    16: (* Transition Delay After Last Bin (Bin 6) Closes *)
        Transition_Timer(IN := TRUE, PT := Step_Delay_Time);
        IF Transition_Timer.Q AND (NOT Discharge_Bin_Coarse[6] AND NOT Discharge_Bin_Fine[6]) THEN
            Transition_Timer(IN := FALSE);
            Step := 7; // Go to post-discharge wait step
        END_IF;

    7: (* Wait 2 Seconds After Closing the Last Bin *)
        Status_Message := 'Settling delay active';
        Completion_Timer(IN := TRUE, PT := Post_Complete_Delay);
        IF Completion_Timer.Q THEN
            Completion_Timer(IN := FALSE);
            Step := 8; // Proceed to reset last weight
        END_IF;
        
    8: (* Reset bin_last_weight to 0 & Complete *)
        bin_last_weight := 0.0;
        Sequence_Complete := TRUE;
        Status_Message := 'Sequence Completed';
        
        IF NOT Start_Button THEN
            Step := 0;
            Sequence_Complete := FALSE;
            Status_Message := 'System Idle';
            (* Reset all actual weights at completion once start is released *)
            FOR i := 1 TO 6 DO
                Actual_Weights[i] := 0.0;
            END_FOR;
        END_IF;
END_CASE;

END_PROGRAM

// PLC_AC500_V3/Application/old_version/Auto_Batching
FUNCTION_BLOCK Auto_Batching
VAR_INPUT
    Start_Button : BOOL;      // Signal to start the batching sequence
    E_Stop_Active : BOOL;     // Emergency Stop active signal
    load_cell_value : REAL;   // Weight value read from load cell
    Discharge_Bin_Feedback : ARRAY[1..6] OF BOOL; // Physical valve feedbacks
END_VAR
VAR_OUTPUT
    Auto_Bin : ARRAY[1..6] OF BOOL; // Motor/valve control outputs
    Actual_Weights : ARRAY[1..6] OF REAL; // Actual weight poured per silo
    Sequence_Complete : BOOL;  // Batch complete flag
END_VAR
VAR
    Step : INT := 0;          // State machine index (0: Idle, 1..6: Bins, 7: Delay, 8: Reset)
    bin_last_weight : REAL;   // Baseline weight on the load cell before starting current bin
    actual_bin : REAL;        // Current weight added from active bin
    target_act_bin : REAL;    // Target weight to add from the active bin
    bin_set_value : REAL;     // Setpoint weight for current active step
    
    (* Bin Mapping for 6 Auto Bins *)
    (* Maps physical Silo 1..6 to Material Index 1..20 *)
    Bin_Material_Index : ARRAY[1..6] OF INT := [
        1,   // Bin 1 maps to Material 1 (50.0 kg)
        2,   // Bin 2 maps to Material 2 (15.0 kg)
        0,   // Bin 3 is 0 (SKIPPED)
        4,   // Bin 4 maps to Material 4 (31.0 kg)
        5,   // Bin 5 maps to Material 5 (150.0 kg)
        6    // Bin 6 maps to Material 6 (10.0 kg)
    ];
    
    Mat_Idx : INT;
    i : INT;                  // General loop index
    
    (* TIMERS FOR TRANSITIONS & DELAYS *)
    Transition_Timer : TON;
    Completion_Timer : TON;
    Step_Delay_Time : TIME := T#2S;
    Post_Complete_Delay : TIME := T#2S;
    
    (* SELF-CONTAINED SIMULATION VARIABLES *)
    Simulation_Mode : BOOL := TRUE;
    Sim_Rate : REAL := 10.0;            // Simulated pouring speed (10.0 kg/s)
    Sim_Timer : TON;
    Start_Sim_Weight : REAL;
    Discharge_Active : BOOL;
END_VAR

(* Cumulative Gain-in-Weight Auto Batching FB *)

(* 1. SELF-CONTAINED SIMULATION WEIGHT MANAGEMENT *)
IF Simulation_Mode THEN
    (* Reset simulation to baseline (e.g. 2.0 kg) *)
    IF Step = 0 AND NOT Start_Button AND NOT Sequence_Complete THEN
        load_cell_value := 2.0;
        bin_last_weight := 2.0;
        Start_Sim_Weight := 2.0;
        Sim_Timer(IN := FALSE);
    END_IF;
    
    (* Check if any valve is actively discharging *)
    Discharge_Active := FALSE;
    IF Step >= 1 AND Step <= 6 THEN
        Discharge_Active := Auto_Bin[Step];
    END_IF;
    
    (* Simulate weight gain on the load cell *)
    IF Discharge_Active THEN
        Sim_Timer(IN := TRUE, PT := T#1000S);
        load_cell_value := Start_Sim_Weight + (TIME_TO_REAL(Sim_Timer.ET) / 1000.0) * Sim_Rate;
    ELSE
        Sim_Timer(IN := FALSE);
        Start_Sim_Weight := load_cell_value;
    END_IF;
END_IF;


(* 2. EMERGENCY STOP LOGIC *)
IF E_Stop_Active THEN
    FOR i := 1 TO 6 DO
        Auto_Bin[i] := FALSE;
        Actual_Weights[i] := 0.0;
    END_FOR;
    Sequence_Complete := FALSE;
    Step := 0;
    Transition_Timer(IN := FALSE);
    Completion_Timer(IN := FALSE);
    RETURN;
END_IF;


(* 3. RECIPE SEQUENCE START *)
IF Step = 0 AND Start_Button THEN
    Step := 1;
    bin_last_weight := load_cell_value;
    Sequence_Complete := FALSE;
    (* Clear actual weights on start *)
    FOR i := 1 TO 6 DO
        Actual_Weights[i] := 0.0;
    END_FOR;
END_IF;


(* 4. SEQUENCE CONTROL STATE MACHINE *)
CASE Step OF
    1..6: (* Discharging Silos 1 to 6 *)
        Mat_Idx := Bin_Material_Index[Step];
        
        IF Mat_Idx = 0 THEN
            (* Skip this bin instantly *)
            Step := Step + 1;
        ELSE
            (* Fetch target weight from global Recipe_Weights array *)
            bin_set_value := GVL.Recipe_Weights[Mat_Idx];
            target_act_bin := bin_set_value;
            
            (* Calculate weight added by current active bin *)
            actual_bin := load_cell_value - bin_last_weight;
            
            (* Update the actual weight in the array for the active bin *)
            Actual_Weights[Step] := actual_bin;
            
            (* Open discharge output valve *)
            Auto_Bin[Step] := TRUE;
            
            (* Check if target weight has been achieved *)
            IF actual_bin >= target_act_bin THEN
                Auto_Bin[Step] := FALSE;
                
                (* Set new baseline for the next step *)
                bin_last_weight := load_cell_value;
                
                (* Go to transition delay *)
                Step := 10 + Step; // Offset to separate transition states
            END_IF;
        END_IF;

    11..15: (* Transition Delays (Between Bins) *)
        Transition_Timer(IN := TRUE, PT := Step_Delay_Time);
        IF Transition_Timer.Q AND (NOT Auto_Bin[Step - 10] OR NOT Discharge_Bin_Feedback[Step - 10]) THEN
            Transition_Timer(IN := FALSE);
            Step := (Step - 10) + 1; // Advance to next bin
        END_IF;
        
    16: (* Transition Delay After Last Bin (Bin 6) Closes *)
        Transition_Timer(IN := TRUE, PT := Step_Delay_Time);
        IF Transition_Timer.Q AND (NOT Auto_Bin[6] OR NOT Discharge_Bin_Feedback[6]) THEN
            Transition_Timer(IN := FALSE);
            Step := 7; // Go to post-discharge wait step
        END_IF;

    7: (* Wait 2 Seconds After Closing the Last Bin *)
        Completion_Timer(IN := TRUE, PT := Post_Complete_Delay);
        IF Completion_Timer.Q THEN
            Completion_Timer(IN := FALSE);
            Step := 8; // Proceed to reset last weight
        END_IF;
        
    8: (* Reset bin_last_weight to 0 & Complete *)
        bin_last_weight := 0.0;
        Sequence_Complete := TRUE;
        
        IF NOT Start_Button THEN
            Step := 0;
            Sequence_Complete := FALSE;
            (* Reset all actual weights at completion once start is released *)
            FOR i := 1 TO 6 DO
                Actual_Weights[i] := 0.0;
            END_FOR;
        END_IF;
END_CASE;

END_FUNCTION_BLOCK

// PLC_AC500_V3/Application/old_version/Manual_Batching
FUNCTION_BLOCK Manual_Batching
VAR_INPUT
    Start_Button : BOOL;      // Signal to start the batching sequence
    E_Stop_Active : BOOL;     // Emergency Stop active signal
    load_cell_value : REAL;   // Weight value read from load cell
END_VAR
VAR_OUTPUT
    Manual_Bin : ARRAY[1..10] OF BOOL; // Prompts/indicators for Bins 7..16
    Actual_Weights : ARRAY[1..10] OF REAL; // Actual weight poured per silo
    Sequence_Complete : BOOL;  // Batch complete flag
END_VAR
VAR
    Step : INT := 0;          // State machine index (0: Idle, 1..10: Bins, 11..20: Delays, 30: Settling, 40: Complete)
    bin_last_weight : REAL;   // Baseline weight on the load cell before starting current bin
    actual_bin : REAL;        // Current weight added from active bin
    target_act_bin : REAL;    // Target weight to add from the active bin
    bin_set_value : REAL;     // Setpoint weight for current active step
    
    (* Bin Mapping for 10 Manual Bins *)
    (* Maps physical manual Silo 7..16 to Material Index 1..20 *)
    Bin_Manual_Index : ARRAY[1..10] OF INT := [
        7,    // Silo 7 maps to Material 7 (12.0 kg)
        8,    // Silo 8 maps to Material 8 (8.0 kg)
        0,    // Silo 9 is 0 (SKIPPED)
        10,   // Silo 10 maps to Material 10 (5.0 kg)
        11,   // Silo 11 maps to Material 11 (18.0 kg)
        12,   // Silo 12 maps to Material 12 (22.0 kg)
        13,   // Silo 13 maps to Material 13 (30.0 kg)
        14,   // Silo 14 maps to Material 14 (14.0 kg)
        15,   // Silo 15 maps to Material 15 (9.0 kg)
        16    // Silo 16 maps to Material 16 (11.0 kg)
    ];
    
    Mat_Idx : INT;
    i : INT;                  // General loop index
    
    (* TIMERS FOR TRANSITIONS & DELAYS *)
    Transition_Timer : TON;
    Completion_Timer : TON;
    Step_Delay_Time : TIME := T#2S;
    Post_Complete_Delay : TIME := T#2S;
    
    (* SELF-CONTAINED SIMULATION VARIABLES *)
    Simulation_Mode : BOOL := TRUE;
    Sim_Rate : REAL := 10.0;            // Simulated pouring speed (10.0 kg/s)
    Sim_Timer : TON;
    Start_Sim_Weight : REAL;
    Discharge_Active : BOOL;
END_VAR

(* Cumulative Gain-in-Weight Manual Batching FB (Simulates Operator Pouring) *)

(* 1. SIMULATION WEIGHT MANAGEMENT *)
IF Simulation_Mode THEN
    (* Reset simulation to baseline (e.g. 2.0 kg) *)
    IF Step = 0 AND NOT Start_Button AND NOT Sequence_Complete THEN
        load_cell_value := 2.0;
        bin_last_weight := 2.0;
        Start_Sim_Weight := 2.0;
        Sim_Timer(IN := FALSE);
    END_IF;
    
    (* Check if operator is actively pouring *)
    Discharge_Active := FALSE;
    IF Step >= 1 AND Step <= 10 THEN
        Discharge_Active := Manual_Bin[Step];
    END_IF;
    
    (* Simulate weight gain on the load cell *)
    IF Discharge_Active THEN
        Sim_Timer(IN := TRUE, PT := T#1000S);
        load_cell_value := Start_Sim_Weight + (TIME_TO_REAL(Sim_Timer.ET) / 1000.0) * Sim_Rate;
    ELSE
        Sim_Timer(IN := FALSE);
        Start_Sim_Weight := load_cell_value;
    END_IF;
END_IF;


(* 2. EMERGENCY STOP LOGIC *)
IF E_Stop_Active THEN
    FOR i := 1 TO 10 DO
        Manual_Bin[i] := FALSE;
        Actual_Weights[i] := 0.0;
    END_FOR;
    Sequence_Complete := FALSE;
    Step := 0;
    Transition_Timer(IN := FALSE);
    Completion_Timer(IN := FALSE);
    RETURN;
END_IF;


(* 3. RECIPE SEQUENCE START *)
IF Step = 0 AND Start_Button THEN
    Step := 1;
    bin_last_weight := load_cell_value;
    Sequence_Complete := FALSE;
    (* Clear actual weights on start *)
    FOR i := 1 TO 10 DO
        Actual_Weights[i] := 0.0;
    END_FOR;
END_IF;


(* 4. SEQUENCE CONTROL STATE MACHINE *)
CASE Step OF
    1..10: (* Prompts Silos 7 to 16 *)
        Mat_Idx := Bin_Manual_Index[Step];
        
        IF Mat_Idx = 0 THEN
            (* Skip this bin instantly *)
            Step := Step + 1;
        ELSE
            (* Fetch target weight from global Recipe_Weights array *)
            bin_set_value := GVL.Recipe_Weights[Mat_Idx];
            target_act_bin := bin_set_value;
            
            (* Calculate weight added by current active bin *)
            actual_bin := load_cell_value - bin_last_weight;
            
            (* Update the actual weight in the array for the active bin *)
            Actual_Weights[Step] := actual_bin;
            
            (* Prompt operator indicator active *)
            Manual_Bin[Step] := TRUE;
            
            (* Check if target weight has been achieved *)
            IF actual_bin >= target_act_bin THEN
                Manual_Bin[Step] := FALSE;
                
                (* Set new baseline for the next step *)
                bin_last_weight := load_cell_value;
                
                (* Go to transition delay *)
                Step := 10 + Step; // Offset to separate transition states
            END_IF;
        END_IF;

    11..19: (* Transition Delays (Between Bins) *)
        Transition_Timer(IN := TRUE, PT := Step_Delay_Time);
        IF Transition_Timer.Q THEN
            Transition_Timer(IN := FALSE);
            Step := (Step - 10) + 1; // Advance to next bin
        END_IF;
        
    20: (* Transition Delay After Last Bin (Bin 10) Closes *)
        Transition_Timer(IN := TRUE, PT := Step_Delay_Time);
        IF Transition_Timer.Q THEN
            Transition_Timer(IN := FALSE);
            Step := 30; // Go to post-discharge wait step (State 30)
        END_IF;

    30: (* Wait 2 Seconds After Closing the Last Bin *)
        Completion_Timer(IN := TRUE, PT := Post_Complete_Delay);
        IF Completion_Timer.Q THEN
            Completion_Timer(IN := FALSE);
            Step := 40; // Proceed to reset last weight (State 40)
        END_IF;
        
    40: (* Reset bin_last_weight to 0 & Complete *)
        bin_last_weight := 0.0;
        Sequence_Complete := TRUE;
        
        IF NOT Start_Button THEN
            Step := 0;
            Sequence_Complete := FALSE;
            (* Reset all actual weights at completion once start is released *)
            FOR i := 1 TO 10 DO
                Actual_Weights[i] := 0.0;
            END_FOR;
        END_IF;
END_CASE;

END_FUNCTION_BLOCK

// PLC_AC500_V3/Application/old_version/batching6
PROGRAM batching6
VAR
    Auto_Ctrl : Auto_Batching;
    Manual_Ctrl : Manual_Batching;
    
    (* Global Inputs & Toggles *)
    Start_Button : BOOL;
    E_Stop_Active : BOOL;
    
    (* Parallel Weight Feedbacks *)
    load_cell_auto : REAL;
    load_cell_manual : REAL;
    
    (* Process Outputs *)
    Auto_Bin : ARRAY[1..6] OF BOOL;
    Manual_Bin : ARRAY[1..10] OF BOOL;
    
    Auto_Weights : ARRAY[1..6] OF REAL;
    Manual_Weights : ARRAY[1..10] OF REAL;
    
    Auto_Complete : BOOL;
    Manual_Complete : BOOL;
    Sequence_Complete : BOOL;
END_VAR

(* Run Auto & Manual Batching pipelines concurrently in parallel *)

Auto_Ctrl(
    Start_Button := Start_Button,
    E_Stop_Active := E_Stop_Active,
    load_cell_value := load_cell_auto,
    Discharge_Bin_Feedback := ,
    Auto_Bin => Auto_Bin,
    Actual_Weights => Auto_Weights,
    Sequence_Complete => Auto_Complete
);

Manual_Ctrl(
    Start_Button := Start_Button,
    E_Stop_Active := E_Stop_Active,
    load_cell_value := load_cell_manual,
    Manual_Bin => Manual_Bin,
    Actual_Weights => Manual_Weights,
    Sequence_Complete => Manual_Complete
);

(* Global complete once both streams conclude *)
Sequence_Complete := Auto_Complete AND Manual_Complete;

END_PROGRAM

// PLC_AC500_V3/Application/old_version/Auto_Batching_V7
FUNCTION_BLOCK Auto_Batching_V7
VAR_INPUT
    Start_Button : BOOL;      // Signal to start the batching sequence
    E_Stop_Active : BOOL;     // Emergency Stop active signal
    load_cell_value : REAL;   // Weight value read from load cell
    Discharge_Bin_Feedback : ARRAY[1..6] OF BOOL; // Physical valve feedbacks
    Bin_Material_Index : ARRAY[1..6] OF INT;      // Mapped material index inputs
END_VAR
VAR_OUTPUT
    Auto_Bin : ARRAY[1..6] OF BOOL; // Motor/valve control outputs
    Actual_Weights : ARRAY[1..6] OF REAL; // Actual weight poured per silo
    Sequence_Complete : BOOL;  // Batch complete flag
    Active_Material_ID : INT;  // Currently active ingredient ID
    Active_Bin_ID : INT;       // Currently active physical Bin ID (1..6)
END_VAR
VAR
    Step : INT := 0;          // State machine index (0: Idle, 1..6: Bins, 7: Delay, 8: Reset)
    bin_last_weight : REAL;   // Baseline weight on the load cell before starting current bin
    actual_bin : REAL;        // Current weight added from active bin
    target_act_bin : REAL;    // Target weight to add from the active bin
    bin_set_value : REAL;     // Setpoint weight for current active step
    
    Mat_Idx : INT;
    i : INT;                  // General loop index
    
    (* TIMERS FOR TRANSITIONS & DELAYS *)
    Transition_Timer : TON;
    Completion_Timer : TON;
    Step_Delay_Time : TIME := T#2S;
    Post_Complete_Delay : TIME := T#2S;
    
    (* SELF-CONTAINED SIMULATION VARIABLES *)
    Simulation_Mode : BOOL := TRUE;
    Sim_Rate : REAL := 10.0;            // Simulated pouring speed (10.0 kg/s)
    Sim_Timer : TON;
    Start_Sim_Weight : REAL;
    Discharge_Active : BOOL;
END_VAR

(* Cumulative Gain-in-Weight Auto Batching FB V7 *)

(* 1. SELF-CONTAINED SIMULATION WEIGHT MANAGEMENT *)
IF Simulation_Mode THEN
    (* Reset simulation to baseline (e.g. 2.0 kg) *)
    IF Step = 0 AND NOT Start_Button AND NOT Sequence_Complete THEN
        load_cell_value := 2.0;
        bin_last_weight := 2.0;
        Start_Sim_Weight := 2.0;
        Sim_Timer(IN := FALSE);
    END_IF;
    
    (* Check if any valve is actively discharging *)
    Discharge_Active := FALSE;
    IF Step >= 1 AND Step <= 6 THEN
        Discharge_Active := Auto_Bin[Step];
    END_IF;
    
    (* Simulate weight gain on the load cell *)
    IF Discharge_Active THEN
        Sim_Timer(IN := TRUE, PT := T#1000S);
        load_cell_value := Start_Sim_Weight + (TIME_TO_REAL(Sim_Timer.ET) / 1000.0) * Sim_Rate;
    ELSE
        Sim_Timer(IN := FALSE);
        Start_Sim_Weight := load_cell_value;
    END_IF;
END_IF;


(* 2. EMERGENCY STOP LOGIC *)
IF E_Stop_Active THEN
    FOR i := 1 TO 6 DO
        Auto_Bin[i] := FALSE;
        Actual_Weights[i] := 0.0;
    END_FOR;
    Sequence_Complete := FALSE;
    Step := 0;
    Active_Material_ID := 0;
    Active_Bin_ID := 0;
    Transition_Timer(IN := FALSE);
    Completion_Timer(IN := FALSE);
    RETURN;
END_IF;


(* 3. RECIPE SEQUENCE START *)
IF Step = 0 AND Start_Button THEN
    Step := 1;
    bin_last_weight := load_cell_value;
    Sequence_Complete := FALSE;
    (* Clear actual weights on start *)
    FOR i := 1 TO 6 DO
        Actual_Weights[i] := 0.0;
    END_FOR;
END_IF;


(* 4. SEQUENCE CONTROL STATE MACHINE *)
CASE Step OF
    0:
        Active_Material_ID := 0;
        Active_Bin_ID := 0;
        
    1..6: (* Discharging Silos 1 to 6 *)
        Mat_Idx := Bin_Material_Index[Step];
        
        IF Mat_Idx = 0 THEN
            (* Skip this bin instantly *)
            Step := Step + 1;
        ELSE
            (* Fetch target weight from global Recipe_Weights array *)
            bin_set_value := GVL.Recipe_Weights[Mat_Idx];
            target_act_bin := bin_set_value;
            
            (* Calculate weight added by current active bin *)
            actual_bin := load_cell_value - bin_last_weight;
            
            (* Update the actual weight in the array for the active bin *)
            Actual_Weights[Step] := actual_bin;
            
            (* Open discharge output valve *)
            Auto_Bin[Step] := TRUE;
            
            (* Output currently active IDs *)
            Active_Material_ID := Mat_Idx;
            Active_Bin_ID := Step;
            
            (* Check if target weight has been achieved *)
            IF actual_bin >= target_act_bin THEN
                Auto_Bin[Step] := FALSE;
                
                (* Set new baseline for the next step *)
                bin_last_weight := load_cell_value;
                
                (* Go to transition delay *)
                Step := 10 + Step; // Offset to separate transition states
            END_IF;
        END_IF;

    11..15: (* Transition Delays (Between Bins) *)
        Active_Material_ID := 0;
        Active_Bin_ID := 0;
        Transition_Timer(IN := TRUE, PT := Step_Delay_Time);
        IF Transition_Timer.Q AND (NOT Auto_Bin[Step - 10] OR NOT Discharge_Bin_Feedback[Step - 10]) THEN
            Transition_Timer(IN := FALSE);
            Step := (Step - 10) + 1; // Advance to next bin
        END_IF;
        
    16: (* Transition Delay After Last Bin (Bin 6) Closes *)
        Active_Material_ID := 0;
        Active_Bin_ID := 0;
        Transition_Timer(IN := TRUE, PT := Step_Delay_Time);
        IF Transition_Timer.Q AND (NOT Auto_Bin[6] OR NOT Discharge_Bin_Feedback[6]) THEN
            Transition_Timer(IN := FALSE);
            Step := 7; // Go to post-discharge wait step
        END_IF;

    7: (* Wait 2 Seconds After Closing the Last Bin *)
        Active_Material_ID := 0;
        Active_Bin_ID := 0;
        Completion_Timer(IN := TRUE, PT := Post_Complete_Delay);
        IF Completion_Timer.Q THEN
            Completion_Timer(IN := FALSE);
            Step := 8; // Proceed to reset last weight
        END_IF;
        
    8: (* Reset bin_last_weight to 0 & Complete *)
        Active_Material_ID := 0;
        Active_Bin_ID := 0;
        bin_last_weight := 0.0;
        Sequence_Complete := TRUE;
        
        IF NOT Start_Button THEN
            Step := 0;
            Sequence_Complete := FALSE;
            (* Reset all actual weights at completion once start is released *)
            FOR i := 1 TO 6 DO
                Actual_Weights[i] := 0.0;
            END_FOR;
        END_IF;
END_CASE;

END_FUNCTION_BLOCK

// PLC_AC500_V3/Application/old_version/Manual_Batching_V7
FUNCTION_BLOCK Manual_Batching_V7
VAR_INPUT
    Start_Button : BOOL;      // Signal to start the batching sequence
    E_Stop_Active : BOOL;     // Emergency Stop active signal
    load_cell_value : REAL;   // Weight value read from load cell
    Bin_Manual_Index : ARRAY[1..10] OF INT; // Mapped material index inputs
END_VAR
VAR_OUTPUT
    Manual_Bin : ARRAY[1..10] OF BOOL; // Prompts/indicators for Bins 7..16
    Actual_Weights : ARRAY[1..10] OF REAL; // Actual weight poured per silo
    Sequence_Complete : BOOL;  // Batch complete flag
    Active_Material_ID : INT;  // Currently active ingredient ID
    Active_Bin_ID : INT;       // Currently active physical Bin ID (7..16)
END_VAR
VAR
    Step : INT := 0;          // State machine index (0: Idle, 1..10: Bins, 11..20: Delays, 30: Settling, 40: Complete)
    bin_last_weight : REAL;   // Baseline weight on the load cell before starting current bin
    actual_bin : REAL;        // Current weight added from active bin
    target_act_bin : REAL;    // Target weight to add from the active bin
    bin_set_value : REAL;     // Setpoint weight for current active step
    
    Mat_Idx : INT;
    i : INT;                  // General loop index
    
    (* TIMERS FOR TRANSITIONS & DELAYS *)
    Transition_Timer : TON;
    Completion_Timer : TON;
    Step_Delay_Time : TIME := T#2S;
    Post_Complete_Delay : TIME := T#2S;
    
    (* SELF-CONTAINED SIMULATION VARIABLES *)
    Simulation_Mode : BOOL := TRUE;
    Sim_Rate : REAL := 10.0;            // Simulated pouring speed (10.0 kg/s)
    Sim_Timer : TON;
    Start_Sim_Weight : REAL;
    Discharge_Active : BOOL;
END_VAR

(* Cumulative Gain-in-Weight Manual Batching FB V7 *)

(* 1. SIMULATION WEIGHT MANAGEMENT *)
IF Simulation_Mode THEN
    (* Reset simulation to baseline (e.g. 2.0 kg) *)
    IF Step = 0 AND NOT Start_Button AND NOT Sequence_Complete THEN
        load_cell_value := 2.0;
        bin_last_weight := 2.0;
        Start_Sim_Weight := 2.0;
        Sim_Timer(IN := FALSE);
    END_IF;
    
    (* Check if operator is actively pouring *)
    Discharge_Active := FALSE;
    IF Step >= 1 AND Step <= 10 THEN
        Discharge_Active := Manual_Bin[Step];
    END_IF;
    
    (* Simulate weight gain on the load cell *)
    IF Discharge_Active THEN
        Sim_Timer(IN := TRUE, PT := T#1000S);
        load_cell_value := Start_Sim_Weight + (TIME_TO_REAL(Sim_Timer.ET) / 1000.0) * Sim_Rate;
    ELSE
        Sim_Timer(IN := FALSE);
        Start_Sim_Weight := load_cell_value;
    END_IF;
END_IF;


(* 2. EMERGENCY STOP LOGIC *)
IF E_Stop_Active THEN
    FOR i := 1 TO 10 DO
        Manual_Bin[i] := FALSE;
        Actual_Weights[i] := 0.0;
    END_FOR;
    Sequence_Complete := FALSE;
    Step := 0;
    Active_Material_ID := 0;
    Active_Bin_ID := 0;
    Transition_Timer(IN := FALSE);
    Completion_Timer(IN := FALSE);
    RETURN;
END_IF;


(* 3. RECIPE SEQUENCE START *)
IF Step = 0 AND Start_Button THEN
    Step := 1;
    bin_last_weight := load_cell_value;
    Sequence_Complete := FALSE;
    (* Clear actual weights on start *)
    FOR i := 1 TO 10 DO
        Actual_Weights[i] := 0.0;
    END_FOR;
END_IF;


(* 4. SEQUENCE CONTROL STATE MACHINE *)
CASE Step OF
    0:
        Active_Material_ID := 0;
        Active_Bin_ID := 0;
        
    1..10: (* Prompts Silos 7 to 16 *)
        Mat_Idx := Bin_Manual_Index[Step];
        
        IF Mat_Idx = 0 THEN
            (* Skip this bin instantly *)
            Step := Step + 1;
        ELSE
            (* Fetch target weight from global Recipe_Weights array *)
            bin_set_value := GVL.Recipe_Weights[Mat_Idx];
            target_act_bin := bin_set_value;
            
            (* Calculate weight added by current active bin *)
            actual_bin := load_cell_value - bin_last_weight;
            
            (* Update the actual weight in the array for the active bin *)
            Actual_Weights[Step] := actual_bin;
            
            (* Prompt operator indicator active *)
            Manual_Bin[Step] := TRUE;
            
            (* Output currently active IDs (Shift to physical Silo ID 7..16) *)
            Active_Material_ID := Mat_Idx;
            Active_Bin_ID := Step;
            
            (* Check if target weight has been achieved *)
            IF actual_bin >= target_act_bin THEN
                Manual_Bin[Step] := FALSE;
                
                (* Set new baseline for the next step *)
                bin_last_weight := load_cell_value;
                
                (* Go to transition delay *)
                Step := 10 + Step; // Offset to separate transition states
            END_IF;
        END_IF;

    11..19: (* Transition Delays (Between Bins) *)
        Active_Material_ID := 0;
        Active_Bin_ID := 0;
        Transition_Timer(IN := TRUE, PT := Step_Delay_Time);
        IF Transition_Timer.Q THEN
            Transition_Timer(IN := FALSE);
            Step := (Step - 10) + 1; // Advance to next bin
        END_IF;
        
    20: (* Transition Delay After Last Bin (Bin 10) Closes *)
        Active_Material_ID := 0;
        Active_Bin_ID := 0;
        Transition_Timer(IN := TRUE, PT := Step_Delay_Time);
        IF Transition_Timer.Q THEN
            Transition_Timer(IN := FALSE);
            Step := 30; // Go to post-discharge wait step (State 30)
        END_IF;

    30: (* Wait 2 Seconds After Closing the Last Bin *)
        Active_Material_ID := 0;
        Active_Bin_ID := 0;
        Completion_Timer(IN := TRUE, PT := Post_Complete_Delay);
        IF Completion_Timer.Q THEN
            Completion_Timer(IN := FALSE);
            Step := 40; // Proceed to reset last weight (State 40)
        END_IF;
        
    40: (* Reset bin_last_weight to 0 & Complete *)
        Active_Material_ID := 0;
        Active_Bin_ID := 0;
        bin_last_weight := 0.0;
        Sequence_Complete := TRUE;
        
        IF NOT Start_Button THEN
            Step := 0;
            Sequence_Complete := FALSE;
            (* Reset all actual weights at completion once start is released *)
            FOR i := 1 TO 10 DO
                Actual_Weights[i] := 0.0;
            END_FOR;
        END_IF;
END_CASE;

END_FUNCTION_BLOCK

// PLC_AC500_V3/Application/old_version/batching7
PROGRAM batching7
VAR
    Auto_Ctrl : Auto_Batching_V7;
    Manual_Ctrl : Manual_Batching_V7;
    
    (* Global Inputs & Toggles *)
    Start_Button : BOOL;
    E_Stop_Active : BOOL;
    
    (* Parallel Weight Feedbacks *)
    load_cell_auto : REAL;
    load_cell_manual : REAL;
    
    (* Process Outputs *)
    Auto_Bin : ARRAY[1..6] OF BOOL;
    Manual_Bin : ARRAY[1..10] OF BOOL;
    
    Auto_Weights : ARRAY[1..6] OF REAL;
    Manual_Weights : ARRAY[1..10] OF REAL;
    
    Auto_Complete : BOOL;
    Manual_Complete : BOOL;
    Sequence_Complete : BOOL;
    
    (* Cross-Validation *)
    Error_Code : INT := 0; // 0 = OK, 1 = Duplicate Material ID detected
    Status_Message : STRING := 'System Ready';
    
    (* Arrays defined here to allow check before FB execution *)
    Bin_Material_Index : ARRAY[1..6] OF INT := [1, 2, 0, 4, 5, 6];
    Bin_Manual_Index : ARRAY[1..10] OF INT := [7, 8, 0, 10, 11, 12, 13, 14, 15, 16];
    
    (* Active IDs as integer monitors *)
    Auto_Active_Mat : INT;
    Auto_Active_Bin : INT;
    Manual_Active_Mat : INT;
    Manual_Active_Bin : INT;
    
    i : INT;
    j : INT;
    Duplicate_Found : BOOL;
END_VAR

(* 1. CROSS-ARRAY DISTINCT MATERIAL VALIDATION *)
Duplicate_Found := FALSE;
FOR i := 1 TO 6 DO
    IF Bin_Material_Index[i] <> 0 THEN
        FOR j := 1 TO 10 DO
            IF Bin_Material_Index[i] = Bin_Manual_Index[j] THEN
                Duplicate_Found := TRUE;
            END_IF;
        END_FOR;
    END_IF;
END_FOR;

IF Duplicate_Found THEN
    Error_Code := 1;
    Status_Message := 'Error 1: Duplicate Material ID in Auto and Manual tables!';
    
    (* Shut off all outputs and abort execution *)
    FOR i := 1 TO 6 DO Auto_Bin[i] := FALSE; END_FOR;
    FOR i := 1 TO 10 DO Manual_Bin[i] := FALSE; END_FOR;
    
    (* Reset control blocks *)
    Auto_Ctrl(Start_Button := FALSE, E_Stop_Active := TRUE);
    Manual_Ctrl(Start_Button := FALSE, E_Stop_Active := TRUE);
    RETURN;
ELSE
    Error_Code := 0;
END_IF;

(* 2. EXECUTION OF BATCH CONTROLLERS *)
Auto_Ctrl(
    Start_Button := Start_Button,
    E_Stop_Active := E_Stop_Active,
    load_cell_value := load_cell_auto,
    Bin_Material_Index := Bin_Material_Index,
    Auto_Bin => Auto_Bin,
    Actual_Weights => Auto_Weights,
    Sequence_Complete => Auto_Complete,
    Active_Material_ID => Auto_Active_Mat,
    Active_Bin_ID => Auto_Active_Bin
);

Manual_Ctrl(
    Start_Button := Start_Button,
    E_Stop_Active := E_Stop_Active,
    load_cell_value := load_cell_manual,
    Bin_Manual_Index := Bin_Manual_Index,
    Manual_Bin => Manual_Bin,
    Actual_Weights => Manual_Weights,
    Sequence_Complete => Manual_Complete,
    Active_Material_ID => Manual_Active_Mat,
    Active_Bin_ID => Manual_Active_Bin
);

Sequence_Complete := Auto_Complete AND Manual_Complete;

IF Sequence_Complete THEN
    Status_Message := 'Batch Completed';
ELSIF Start_Button THEN
    Status_Message := 'Batch In Progress';
ELSE
    Status_Message := 'System Ready';
END_IF;

END_PROGRAM

// PLC_AC500_V3/Application/old_version/Auto_Batching_V8
FUNCTION_BLOCK Auto_Batching_V8
VAR_INPUT
    Start_Button : BOOL;      // Signal to start the batching sequence
    E_Stop_Active : BOOL;     // Emergency Stop active signal
    Discharge_Bin_Feedback : ARRAY[1..6] OF BOOL; // Physical valve feedbacks
    Auto_Bin_Material_Mapping : ARRAY[1..6] OF INT; // Material index mapping for 6 bins
    Auto_Coarse_To_Fine_speed : ARRAY[1..6] OF REAL; // Cutoff weight thresholds (kg)
END_VAR
VAR_IN_OUT
    load_cell_value : REAL;   // Weight value read/written from load cell
END_VAR
VAR_OUTPUT
    Auto_Bin : ARRAY[1..6] OF BOOL; // Coarse feed valve outputs
    auto_bin_cutoff : ARRAY[1..6] OF BOOL; // Fine feed cutoff trigger indicators
    auto_bin_motor : ARRAY[1..6] OF BOOL; // Main conveyor motor outputs
    Actual_Weights : ARRAY[1..6] OF REAL; // Actual weight poured per silo
    Sequence_Complete : BOOL;  // Batch complete flag
    Active_Material_ID : INT;  // Currently active ingredient ID
    Active_Bin_ID : INT;       // Currently active physical Bin ID (1..6)
    Active_Target_Weight : REAL; // Recipe target weight of active bin
    Error_Code : INT;          // Active error code
    Status_Message : STRING;   // Diagnostic text message
END_VAR
VAR
    Step : INT := 0;          // State machine index (0: Idle, 1..6: Bins, 11..16: Delays, 7: Settling, 8: Complete, 99: Error)
    bin_last_weight : REAL;   // Baseline weight on the load cell before starting current bin
    actual_bin : REAL;        // Current weight added from active bin
    target_act_bin : REAL;    // Target weight to add from the active bin
    bin_set_value : REAL;     // Setpoint weight for current active step
    cutoff_trigger_weight : REAL; // Calculated target threshold weight minus cutoff value
    
    Mat_Idx : INT;
    i : INT;                  // General loop index
    
    (* TIMERS FOR TRANSITIONS & DELAYS *)
    Transition_Timer : TON;
    Completion_Timer : TON;
    Step_Delay_Time : TIME := T#2S;
    Post_Complete_Delay : TIME := T#2S;
    
    (* SELF-CONTAINED SIMULATION VARIABLES *)
    Simulation_Mode : BOOL := TRUE;
    Sim_Rate : REAL := 10.0;            // Simulated pouring speed (10.0 kg/s)
    Sim_Timer : TON;
    Start_Sim_Weight : REAL;
    Discharge_Active : BOOL;
END_VAR

(* Auto Batching FB V8 matching batching7 sequence exactly *)

(* 1. SELF-CONTAINED SIMULATION WEIGHT MANAGEMENT *)
IF Simulation_Mode AND Step <> 99 THEN
    (* Reset simulation to baseline *)
    IF Step = 0 AND NOT Start_Button AND NOT Sequence_Complete THEN
        load_cell_value := 0.0;
        bin_last_weight := 0.0;
        Start_Sim_Weight := 0.0;
        Sim_Timer(IN := FALSE);
    END_IF;
    
    (* Check if any valve is actively discharging *)
    Discharge_Active := FALSE;
    IF Step >= 1 AND Step <= 6 THEN
        Discharge_Active := auto_bin_motor[Step];
    END_IF;
    
    (* Simulate weight gain on the load cell *)
    IF Discharge_Active THEN
        Sim_Timer(IN := TRUE, PT := T#1000S);
        load_cell_value := Start_Sim_Weight + (TIME_TO_REAL(Sim_Timer.ET) / 1000.0) * Sim_Rate;
    ELSE
        Sim_Timer(IN := FALSE);
        Start_Sim_Weight := load_cell_value;
    END_IF;
END_IF;


(* 2. EMERGENCY STOP LOGIC (Error 12) *)
IF E_Stop_Active THEN
    FOR i := 1 TO 6 DO
        Auto_Bin[i] := FALSE;
        auto_bin_cutoff[i] := FALSE;
        auto_bin_motor[i] := FALSE;
    END_FOR;
    Sequence_Complete := FALSE;
    Active_Material_ID := 0;
    Active_Bin_ID := 0;
    Active_Target_Weight := 0.0;
    Error_Code := 12;
    Status_Message := 'Error 12: Emergency Stop Active!';
    Step := 99;
    Transition_Timer(IN := FALSE);
    Completion_Timer(IN := FALSE);
    RETURN;
END_IF;


(* 3. RECIPE SEQUENCE START *)
IF Step = 0 AND Start_Button THEN
    Step := 1;
    bin_last_weight := load_cell_value;
    Sequence_Complete := FALSE;
    Error_Code := 0;
    Status_Message := 'Auto Batch Started';
    Active_Target_Weight := 0.0;
    (* Clear actual weights and outputs on start *)
    FOR i := 1 TO 6 DO
        Actual_Weights[i] := 0.0;
        Auto_Bin[i] := FALSE;
        auto_bin_cutoff[i] := FALSE;
        auto_bin_motor[i] := FALSE;
    END_FOR;
END_IF;


(* 4. SEQUENCE CONTROL STATE MACHINE *)
CASE Step OF
    0:
        Active_Material_ID := 0;
        Active_Bin_ID := 0;
        Active_Target_Weight := 0.0;
        IF Error_Code = 0 THEN Status_Message := 'Auto Idle'; END_IF;
        
    1..6: (* Discharging Silos 1 to 6 *)
        Mat_Idx := Auto_Bin_Material_Mapping[Step];
        
        IF Mat_Idx = 0 THEN
            (* Skip this bin instantly *)
            Step := Step + 1;
        ELSE
            (* Fetch target weight from global Recipe_Weights array *)
            bin_set_value := GVL.Recipe_Weights[Mat_Idx];
            target_act_bin := bin_set_value;
            Active_Target_Weight := target_act_bin;
            
            (* Calculate weight added by current active bin *)
            actual_bin := load_cell_value - bin_last_weight;
            Actual_Weights[Step] := actual_bin;
            
            (* Get cutoff threshold *)
            cutoff_trigger_weight := target_act_bin - Auto_Coarse_To_Fine_speed[Step];
            
            Active_Material_ID := Mat_Idx;
            Active_Bin_ID := Step;
            Status_Message := 'Auto Pouring';
            
            (* COARSE/FINE FEED TRANSITIONS *)
            IF actual_bin < cutoff_trigger_weight THEN
                (* Phase 1: Coarse Feed (Conveyor Motor ON, Main Valve ON, Fine Cutoff OFF) *)
                Auto_Bin[Step] := TRUE;
                auto_bin_cutoff[Step] := FALSE;
                auto_bin_motor[Step] := TRUE;
            ELSIF actual_bin < target_act_bin THEN
                (* Phase 2: Fine Feed (Conveyor Motor ON, Main Valve OFF, Fine Cutoff ON) *)
                Auto_Bin[Step] := FALSE;
                auto_bin_cutoff[Step] := TRUE;
                auto_bin_motor[Step] := TRUE;
            ELSE
                (* Phase 3: Completed (All OFF) *)
                Auto_Bin[Step] := FALSE;
                auto_bin_cutoff[Step] := FALSE;
                auto_bin_motor[Step] := FALSE;
                bin_last_weight := load_cell_value;
                Active_Target_Weight := 0.0;
                Step := 10 + Step; // Offset to separate transition states
            END_IF;
            
            (* RUNTIME CHECKS *)
            (* Check 21 & 22: Scale Limits *)
            IF load_cell_value > 500.0 THEN
                Error_Code := 21;
                Status_Message := 'Error 21: Scale Overloaded!';
                Step := 99;
                RETURN;
            ELSIF load_cell_value < 0.0 THEN
                Error_Code := 22;
                Status_Message := 'Error 22: Scale Underloaded/Fault!';
                Step := 99;
                RETURN;
            END_IF;
        END_IF;

    11..15: (* Transition Delays (Between Bins) *)
        Active_Material_ID := 0;
        Active_Bin_ID := 0;
        Active_Target_Weight := 0.0;
        Status_Message := 'Transition Delay';
        
        Transition_Timer(IN := TRUE, PT := Step_Delay_Time);
        IF Transition_Timer.Q THEN
            Transition_Timer(IN := FALSE);
            Step := (Step - 10) + 1; // Advance to next bin
        END_IF;
        
    16: (* Transition Delay After Last Bin (Bin 6) Closes *)
        Active_Material_ID := 0;
        Active_Bin_ID := 0;
        Active_Target_Weight := 0.0;
        Status_Message := 'Settling Last Bin';
        
        Transition_Timer(IN := TRUE, PT := Step_Delay_Time);
        IF Transition_Timer.Q THEN
            Transition_Timer(IN := FALSE);
            Step := 7; // Go to post-discharge wait step
        END_IF;

    7: (* Wait 2 Seconds After Closing the Last Bin *)
        Active_Material_ID := 0;
        Active_Bin_ID := 0;
        Active_Target_Weight := 0.0;
        Status_Message := 'Settling Delay';
        Completion_Timer(IN := TRUE, PT := Post_Complete_Delay);
        IF Completion_Timer.Q THEN
            Completion_Timer(IN := FALSE);
            Step := 8; // Proceed to reset last weight
        END_IF;
        
    8: (* Reset bin_last_weight to 0 & Complete *)
        Active_Material_ID := 0;
        Active_Bin_ID := 0;
        Active_Target_Weight := 0.0;
        Status_Message := 'Sequence Completed';
        bin_last_weight := 0.0;
        Sequence_Complete := TRUE;
        
        IF NOT Start_Button THEN
            Step := 0;
            Sequence_Complete := FALSE;
            (* Reset all actual weights at completion once start is released *)
            FOR i := 1 TO 6 DO
                Actual_Weights[i] := 0.0;
            END_FOR;
        END_IF;
        
    99: (* Error Abort state *)
        FOR i := 1 TO 6 DO 
            Auto_Bin[i] := FALSE; 
            auto_bin_cutoff[i] := FALSE;
            auto_bin_motor[i] := FALSE;
        END_FOR;
        Active_Material_ID := 0;
        Active_Bin_ID := 0;
        Active_Target_Weight := 0.0;
        IF NOT Start_Button THEN
            Step := 0;
            Error_Code := 0;
            Status_Message := 'Auto Idle';
        END_IF;
END_CASE;

END_FUNCTION_BLOCK

// PLC_AC500_V3/Application/old_version/Manual_Batching_V8
FUNCTION_BLOCK Manual_Batching_V8
VAR_INPUT
    Start_Button : BOOL;      // Signal to start the batching sequence
    E_Stop_Active : BOOL;     // Emergency Stop active signal
    Manual_Bin_Material_Mapping : ARRAY[1..10] OF INT; // Material index mapping for 10 manual silos
    Manual_Coarse_To_Fine_speed : ARRAY[1..10] OF REAL; // Cutoff weight thresholds (kg)
END_VAR
VAR_IN_OUT
    load_cell_value : REAL;   // Weight value read/written from load cell
END_VAR
VAR_OUTPUT
    Manual_Bin : ARRAY[1..10] OF BOOL; // Prompts/indicators for Bins 7..16
    manual_bin_cutoff : ARRAY[1..10] OF BOOL; // Manual pre-cutoff indicators
    manual_bin_motor : ARRAY[1..10] OF BOOL; // Main manual feeder motor outputs
    Actual_Weights : ARRAY[1..10] OF REAL; // Actual weight poured per silo
    Sequence_Complete : BOOL;  // Batch complete flag
    Active_Material_ID : INT;  // Currently active ingredient ID
    Active_Bin_ID : INT;       // Currently active physical Bin ID (7..16)
    Active_Target_Weight : REAL; // Recipe target weight of active bin
    Error_Code : INT;          // Active error code
    Status_Message : STRING;   // Diagnostic text message
END_VAR
VAR
    Step : INT := 0;          // State machine index (0: Idle, 1..10: Bins, 11..20: Delays, 30: Settling, 40: Complete, 99: Error)
    bin_last_weight : REAL;   // Baseline weight on the load cell before starting current bin
    actual_bin : REAL;        // Current weight added from active bin
    target_act_bin : REAL;    // Target weight to add from the active bin
    bin_set_value : REAL;     // Setpoint weight for current active step
    cutoff_trigger_weight : REAL; // Calculated target threshold weight minus cutoff value
    
    Mat_Idx : INT;
    i : INT;                  // General loop index
    
    (* TIMERS FOR TRANSITIONS & DELAYS *)
    Transition_Timer : TON;
    Completion_Timer : TON;
    Step_Delay_Time : TIME := T#2S;
    Post_Complete_Delay : TIME := T#2S;
    
    (* DIAGNOSTIC TIMERS *)
    Operator_Timer : TON;
    
    (* SELF-CONTAINED SIMULATION VARIABLES *)
    Simulation_Mode : BOOL := TRUE;
    Sim_Rate : REAL := 10.0;            // Simulated pouring speed (10.0 kg/s)
    Sim_Timer : TON;
    Start_Sim_Weight : REAL;
    Discharge_Active : BOOL;
END_VAR

(* Manual Batching FB V8 with Diagnostic Error Checks *)

(* 1. SIMULATION WEIGHT MANAGEMENT *)
IF Simulation_Mode AND Step <> 99 THEN
    (* Reset simulation to baseline *)
    IF Step = 0 AND NOT Start_Button AND NOT Sequence_Complete THEN
        load_cell_value := 0.0;
        bin_last_weight := 0.0;
        Start_Sim_Weight := 0.0;
        Sim_Timer(IN := FALSE);
    END_IF;
    
    (* Check if operator is actively pouring *)
    Discharge_Active := FALSE;
    IF Step >= 1 AND Step <= 10 THEN
        Discharge_Active := manual_bin_motor[Step];
    END_IF;
    
    (* Simulate weight gain on the load cell *)
    IF Discharge_Active THEN
        Sim_Timer(IN := TRUE, PT := T#1000S);
        load_cell_value := Start_Sim_Weight + (TIME_TO_REAL(Sim_Timer.ET) / 1000.0) * Sim_Rate;
    ELSE
        Sim_Timer(IN := FALSE);
        Start_Sim_Weight := load_cell_value;
    END_IF;
END_IF;


(* 2. EMERGENCY STOP LOGIC (Error 12) *)
IF E_Stop_Active THEN
    FOR i := 1 TO 10 DO
        Manual_Bin[i] := FALSE;
        manual_bin_cutoff[i] := FALSE;
        manual_bin_motor[i] := FALSE;
    END_FOR;
    Sequence_Complete := FALSE;
    Active_Material_ID := 0;
    Active_Bin_ID := 0;
    Active_Target_Weight := 0.0;
    Error_Code := 12;
    Status_Message := 'Error 12: Emergency Stop Active!';
    Step := 99;
    Transition_Timer(IN := FALSE);
    Completion_Timer(IN := FALSE);
    RETURN;
END_IF;


(* 3. RECIPE SEQUENCE START *)
IF Step = 0 AND Start_Button THEN
    Step := 1;
    bin_last_weight := load_cell_value;
    Sequence_Complete := FALSE;
    Error_Code := 0;
    Status_Message := 'Manual Batch Started';
    Active_Target_Weight := 0.0;
    (* Clear actual weights on start *)
    FOR i := 1 TO 10 DO
        Actual_Weights[i] := 0.0;
        Manual_Bin[i] := FALSE;
        manual_bin_cutoff[i] := FALSE;
        manual_bin_motor[i] := FALSE;
    END_FOR;
END_IF;


(* 4. SEQUENCE CONTROL STATE MACHINE *)
CASE Step OF
    0:
        Active_Material_ID := 0;
        Active_Bin_ID := 0;
        Active_Target_Weight := 0.0;
        IF Error_Code = 0 THEN Status_Message := 'Manual Idle'; END_IF;
        
    1..10: (* Prompts Silos 7 to 16 *)
        Mat_Idx := Manual_Bin_Material_Mapping[Step];
        
        IF Mat_Idx = 0 THEN
            (* Skip this bin instantly *)
            Step := Step + 1;
        ELSE
            (* Fetch target weight from global Recipe_Weights array *)
            bin_set_value := GVL.Recipe_Weights[Mat_Idx];
            target_act_bin := bin_set_value;
            Active_Target_Weight := target_act_bin;
            
            (* Calculate weight added by current active bin *)
            actual_bin := load_cell_value - bin_last_weight;
            Actual_Weights[Step] := actual_bin;
            
            (* Get cutoff threshold *)
            cutoff_trigger_weight := target_act_bin - Manual_Coarse_To_Fine_speed[Step];
            
            Active_Material_ID := Mat_Idx;
            Active_Bin_ID := Step;
            Status_Message := 'Manual Pouring Active';
            
            (* COARSE/FINE FEED TRANSITIONS *)
            IF actual_bin < cutoff_trigger_weight THEN
                (* Phase 1: Coarse Feed (Motor ON, Prompt ON, Cutoff OFF) *)
                Manual_Bin[Step] := TRUE;
                manual_bin_cutoff[Step] := FALSE;
                manual_bin_motor[Step] := TRUE;
            ELSIF actual_bin < target_act_bin THEN
                (* Phase 2: Fine Feed (Motor ON, Prompt OFF, Cutoff ON) *)
                Manual_Bin[Step] := FALSE;
                manual_bin_cutoff[Step] := TRUE;
                manual_bin_motor[Step] := TRUE;
            ELSE
                (* Phase 3: Completed (All OFF) *)
                Manual_Bin[Step] := FALSE;
                manual_bin_cutoff[Step] := FALSE;
                manual_bin_motor[Step] := FALSE;
                bin_last_weight := load_cell_value;
                Active_Target_Weight := 0.0;
                Step := 10 + Step; // Offset to separate transition states
            END_IF;
            
            (* RUNTIME CHECKS *)
            (* Check 21 & 22: Scale Limits *)
            IF load_cell_value > 500.0 THEN
                Error_Code := 21;
                Status_Message := 'Error 21: Scale Overloaded!';
                Step := 99;
                RETURN;
            ELSIF load_cell_value < 0.0 THEN
                Error_Code := 22;
                Status_Message := 'Error 22: Scale Underloaded/Fault!';
                Step := 99;
                RETURN;
            END_IF;
            
            (* Check 30: Operator Timeout *)
            Operator_Timer(IN := manual_bin_motor[Step], PT := T#300S);
            IF Operator_Timer.Q THEN
                Error_Code := 30;
                Status_Message := 'Error 30: Manual Operator Timeout!';
                Step := 99;
                RETURN;
            END_IF;
        END_IF;

    11..19: (* Transition Delays (Between Bins) *)
        Active_Material_ID := 0;
        Active_Bin_ID := 0;
        Active_Target_Weight := 0.0;
        Status_Message := 'Transition Delay';
        Transition_Timer(IN := TRUE, PT := Step_Delay_Time);
        IF Transition_Timer.Q THEN
            Transition_Timer(IN := FALSE);
            Step := (Step - 10) + 1; // Advance to next bin
        END_IF;
        
    20: (* Transition Delay After Last Bin (Bin 10) Closes *)
        Active_Material_ID := 0;
        Active_Bin_ID := 0;
        Active_Target_Weight := 0.0;
        Status_Message := 'Settling Last Bin';
        Transition_Timer(IN := TRUE, PT := Step_Delay_Time);
        IF Transition_Timer.Q THEN
            Transition_Timer(IN := FALSE);
            Step := 30; // Go to post-discharge wait step (State 30)
        END_IF;

    30: (* Wait 2 Seconds After Closing the Last Bin *)
        Active_Material_ID := 0;
        Active_Bin_ID := 0;
        Active_Target_Weight := 0.0;
        Status_Message := 'Settling Delay';
        Completion_Timer(IN := TRUE, PT := Post_Complete_Delay);
        IF Completion_Timer.Q THEN
            Completion_Timer(IN := FALSE);
            Step := 40; // Proceed to reset last weight (State 40)
        END_IF;
        
    40: (* Reset bin_last_weight to 0 & Complete *)
        Active_Material_ID := 0;
        Active_Bin_ID := 0;
        Active_Target_Weight := 0.0;
        Status_Message := 'Sequence Completed';
        bin_last_weight := 0.0;
        Sequence_Complete := TRUE;
        
        IF NOT Start_Button THEN
            Step := 0;
            Sequence_Complete := FALSE;
            (* Reset all actual weights at completion once start is released *)
            FOR i := 1 TO 10 DO
                Actual_Weights[i] := 0.0;
            END_FOR;
        END_IF;
        
    99: (* Error Abort state *)
        FOR i := 1 TO 10 DO 
            Manual_Bin[i] := FALSE;
            manual_bin_cutoff[i] := FALSE;
            manual_bin_motor[i] := FALSE;
        END_FOR;
        Active_Material_ID := 0;
        Active_Bin_ID := 0;
        Active_Target_Weight := 0.0;
        IF NOT Start_Button THEN
            Step := 0;
            Error_Code := 0;
            Status_Message := 'Manual Idle';
        END_IF;
END_CASE;

END_FUNCTION_BLOCK

// PLC_AC500_V3/Application/old_version/batching8
PROGRAM batching8
VAR
    Auto_Ctrl : Auto_Batching_V8;
    Manual_Ctrl : Manual_Batching_V8;
    
    (* Global Inputs & Toggles *)
    Start_Button : BOOL;
    E_Stop_Active : BOOL;
    
    (* Parallel Weight Feedbacks *)
    load_cell_auto : REAL;
    load_cell_manual : REAL;
    
    (* Sub-Block Diagnostic Indicators - Ordered exactly below loadcell *)
    Auto_Active_Mat : INT;
    Auto_Active_Bin : INT;
    Auto_Active_Target : REAL; // Active Target Weight for Auto (displays GVL setpoint)
    Auto_Err : INT;
    Auto_Msg : STRING;
    
    Manual_Active_Mat : INT;
    Manual_Active_Bin : INT;
    Manual_Active_Target : REAL; // Active Target Weight for Manual (displays GVL setpoint)
    Manual_Err : INT;
    Manual_Msg : STRING;
    
    (* Process Outputs *)
    Auto_Bin : ARRAY[1..6] OF BOOL; // Valve control outputs (Coarse)
    auto_bin_cutoff : ARRAY[1..6] OF BOOL; // Cutoff indicators (Fine)
    auto_bin_motor : ARRAY[1..6] OF BOOL; // Conveyor/feeder motor outputs
    
    Manual_Bin : ARRAY[1..10] OF BOOL; // Prompt indicators (Coarse)
    manual_bin_cutoff : ARRAY[1..10] OF BOOL; // Cutoff indicators (Fine)
    manual_bin_motor : ARRAY[1..10] OF BOOL; // Conveyor/feeder motor outputs
    
    Auto_Weights : ARRAY[1..6] OF REAL;
    Manual_Weights : ARRAY[1..10] OF REAL;
    
    Auto_Complete : BOOL;
    Manual_Complete : BOOL;
    Sequence_Complete : BOOL;
    
    (* Diagnostics & Interlocks *)
    Error_Code : INT := 0;
    Status_Message : STRING := 'System Ready';
    
    (* Array Configurations & Mapping - Renamed for clarity *)
    Auto_Bin_Material_Mapping : ARRAY[1..6] OF INT := [1, 2, 0, 4, 5, 6];
    Manual_Bin_Material_Mapping : ARRAY[1..10] OF INT := [7, 8, 0, 10, 11, 12, 13, 14, 15, 16];
    Auto_Coarse_To_Fine_speed : ARRAY[1..6] OF REAL := [2.0, 1.5, 0.0, 3.0, 5.0, 1.0]; // Cutoff margins (kg)
    Manual_Coarse_To_Fine_speed : ARRAY[1..10] OF REAL := [2.0, 1.5, 0.0, 3.0, 5.0, 1.0, 2.0, 2.0, 2.0, 2.0];
    
    i : INT;
    j : INT;
    Duplicate_Found : BOOL;
    Invalid_Material_Range : BOOL;
    Zero_Target_Found : BOOL;
    Conf_Err_Id : INT;
END_VAR

(* 1. STARTUP CONFIGURATION CHECKS *)
Duplicate_Found := FALSE;
Invalid_Material_Range := FALSE;
Zero_Target_Found := FALSE;

FOR i := 1 TO 6 DO
    (* Check 2: Out of Range (Auto) *)
    IF Auto_Bin_Material_Mapping[i] < 0 OR Auto_Bin_Material_Mapping[i] > 20 THEN
        Invalid_Material_Range := TRUE;
    END_IF;
    
    (* Check 3: Zero Target (Auto) *)
    IF Auto_Bin_Material_Mapping[i] <> 0 AND Auto_Bin_Material_Mapping[i] <= 20 THEN
        IF GVL.Recipe_Weights[Auto_Bin_Material_Mapping[i]] = 0.0 THEN
            Zero_Target_Found := TRUE;
        END_IF;
    END_IF;
    
    (* Check 1: Duplicate Cross-Array Material ID *)
    IF Auto_Bin_Material_Mapping[i] <> 0 AND Auto_Bin_Material_Mapping[i] <= 20 THEN
        FOR j := 1 TO 10 DO
            IF Auto_Bin_Material_Mapping[i] = Manual_Bin_Material_Mapping[j] THEN
                Duplicate_Found := TRUE;
            END_IF;
        END_FOR;
    END_IF;
END_FOR;

FOR j := 1 TO 10 DO
    (* Check 2: Out of Range (Manual) *)
    IF Manual_Bin_Material_Mapping[j] < 0 OR Manual_Bin_Material_Mapping[j] > 20 THEN
        Invalid_Material_Range := TRUE;
    END_IF;
    
    (* Check 3: Zero Target (Manual) *)
    IF Manual_Bin_Material_Mapping[j] <> 0 AND Manual_Bin_Material_Mapping[j] <= 20 THEN
        IF GVL.Recipe_Weights[Manual_Bin_Material_Mapping[j]] = 0.0 THEN
            Zero_Target_Found := TRUE;
        END_IF;
    END_IF;
END_FOR;

(* Configuration Error Resolution *)
IF Duplicate_Found THEN
    Error_Code := 1;
    Status_Message := 'Error 1: Duplicate Material ID mapped in Auto and Manual!';
ELSIF Invalid_Material_Range THEN
    Error_Code := 2;
    Status_Message := 'Error 2: Material Index configuration out of range (1..20)!';
ELSIF Zero_Target_Found THEN
    Error_Code := 3;
    Status_Message := 'Error 3: Configured Material ID has a 0.0 kg target weight!';
ELSE
    IF Error_Code <= 3 THEN
        Error_Code := 0;
    END_IF;
END_IF;

(* Abort sequences if a configuration error exists *)
IF Error_Code >= 1 AND Error_Code <= 3 THEN
    FOR i := 1 TO 6 DO Auto_Bin[i] := FALSE; auto_bin_cutoff[i] := FALSE; auto_bin_motor[i] := FALSE; END_FOR;
    FOR i := 1 TO 10 DO Manual_Bin[i] := FALSE; manual_bin_cutoff[i] := FALSE; manual_bin_motor[i] := FALSE; END_FOR;
    Auto_Ctrl(Start_Button := FALSE, E_Stop_Active := TRUE, load_cell_value := load_cell_auto);
    Manual_Ctrl(Start_Button := FALSE, E_Stop_Active := TRUE, load_cell_value := load_cell_manual);
    Auto_Active_Target := 0.0;
    Manual_Active_Target := 0.0;
    RETURN;
END_IF;


(* 2. CONCURRENT EXECUTION OF FB INSTANCES *)
Auto_Ctrl(
    Start_Button := Start_Button,
    E_Stop_Active := E_Stop_Active,
    load_cell_value := load_cell_auto,
    Auto_Bin_Material_Mapping := Auto_Bin_Material_Mapping,
    Auto_Coarse_To_Fine_speed := Auto_Coarse_To_Fine_speed,
    Auto_Bin => Auto_Bin,
    auto_bin_cutoff => auto_bin_cutoff,
    auto_bin_motor => auto_bin_motor,
    Actual_Weights => Auto_Weights,
    Sequence_Complete => Auto_Complete,
    Active_Material_ID => Auto_Active_Mat,
    Active_Bin_ID => Auto_Active_Bin,
    Active_Target_Weight => Auto_Active_Target,
    Error_Code => Auto_Err,
    Status_Message => Auto_Msg
);

Manual_Ctrl(
    Start_Button := Start_Button,
    E_Stop_Active := E_Stop_Active,
    load_cell_value := load_cell_manual,
    Manual_Bin_Material_Mapping := Manual_Bin_Material_Mapping,
    Manual_Coarse_To_Fine_speed := Manual_Coarse_To_Fine_speed,
    Manual_Bin => Manual_Bin,
    manual_bin_cutoff => manual_bin_cutoff,
    manual_bin_motor => manual_bin_motor,
    Actual_Weights => Manual_Weights,
    Sequence_Complete => Manual_Complete,
    Active_Material_ID => Manual_Active_Mat,
    Active_Bin_ID => Manual_Active_Bin,
    Active_Target_Weight => Manual_Active_Target,
    Error_Code => Manual_Err,
    Status_Message => Manual_Msg
);

(* Runtime Error Mapping & Aggregation *)
IF Auto_Err <> 0 THEN
    Error_Code := Auto_Err;
    Status_Message := CONCAT('Auto Error: ', Auto_Msg);
ELSIF Manual_Err <> 0 THEN
    Error_Code := Manual_Err;
    Status_Message := CONCAT('Manual Error: ', Manual_Msg);
ELSE
    Error_Code := 0;
    
    Sequence_Complete := Auto_Complete AND Manual_Complete;
    IF Sequence_Complete THEN
        Status_Message := 'Batch Sequence Completed';
    ELSIF Start_Button THEN
        Status_Message := 'Batch Sequence Running';
    ELSE
        Status_Message := 'System Ready';
    END_IF;
END_IF;

END_PROGRAM

// PLC_AC500_V3/Application/old_version/Auto_Batching_V9
FUNCTION_BLOCK Auto_Batching_V9
VAR_INPUT
    Start_Button : BOOL;      // Signal to start the batching sequence
    E_Stop_Active : BOOL;     // Emergency Stop active signal
    Discharge_Bin_Feedback : ARRAY[1..6] OF BOOL; // Physical valve feedbacks
    Auto_Bin_Material_Mapping : ARRAY[1..6] OF INT; // Material index mapping for 6 bins
    Auto_Coarse_To_Fine_speed : ARRAY[1..6] OF REAL; // Cutoff weight thresholds (kg)
    Auto_Bin_Tolerance : ARRAY[1..6] OF REAL; // Tolerance weight offset values (kg)
END_VAR
VAR_IN_OUT
    load_cell_value : REAL;   // Weight value read/written from load cell
END_VAR
VAR_OUTPUT
    Auto_Bin : ARRAY[1..6] OF BOOL; // Coarse feed valve outputs
    auto_bin_cutoff : ARRAY[1..6] OF BOOL; // Fine feed cutoff trigger indicators
    auto_bin_motor : ARRAY[1..6] OF BOOL; // Main conveyor motor outputs
    Actual_Weights : ARRAY[1..6] OF REAL; // Actual weight poured per silo
    Sequence_Complete : BOOL;  // Batch complete flag
    Active_Material_ID : INT;  // Currently active ingredient ID
    Active_Bin_ID : INT;       // Currently active physical Bin ID (1..6)
    Active_Target_Weight : REAL; // Recipe target weight of active bin (with tolerance applied)
    Error_Code : INT;          // Active error code
    Status_Message : STRING;   // Diagnostic text message
END_VAR
VAR
    Step : INT := 0;          // State machine index (0: Idle, 1..6: Bins, 11..16: Delays, 7: Settling, 8: Complete, 99: Error)
    bin_last_weight : REAL;   // Baseline weight on the load cell before starting current bin
    actual_bin : REAL;        // Current weight added from active bin
    target_act_bin : REAL;    // Effective target weight to add from the active bin (GVL target - Tolerance)
    bin_set_value : REAL;     // Setpoint weight looked up from GVL
    cutoff_trigger_weight : REAL; // Calculated trigger weight (target - Tolerance - Cutoff)
    
    Mat_Idx : INT;
    i : INT;                  // General loop index
    
    (* TIMERS FOR TRANSITIONS & DELAYS *)
    Transition_Timer : TON;
    Completion_Timer : TON;
    Step_Delay_Time : TIME := T#2S;
    Post_Complete_Delay : TIME := T#2S;
    
    (* SELF-CONTAINED SIMULATION VARIABLES *)
    Simulation_Mode : BOOL := TRUE;
    Sim_Rate : REAL := 10.0;            // Simulated pouring speed (10.0 kg/s)
    Sim_Timer : TON;
    Start_Sim_Weight : REAL;
    Discharge_Active : BOOL;
END_VAR

(* Auto Batching FB V9 with Tolerance Logic *)

(* 1. SELF-CONTAINED SIMULATION WEIGHT MANAGEMENT *)
IF Simulation_Mode AND Step <> 99 THEN
    (* Reset simulation to baseline *)
    IF Step = 0 AND NOT Start_Button AND NOT Sequence_Complete THEN
        load_cell_value := 0.0;
        bin_last_weight := 0.0;
        Start_Sim_Weight := 0.0;
        Sim_Timer(IN := FALSE);
    END_IF;
    
    (* Check if any valve is actively discharging *)
    Discharge_Active := FALSE;
    IF Step >= 1 AND Step <= 6 THEN
        Discharge_Active := auto_bin_motor[Step];
    END_IF;
    
    (* Simulate weight gain on the load cell *)
    IF Discharge_Active THEN
        Sim_Timer(IN := TRUE, PT := T#1000S);
        load_cell_value := Start_Sim_Weight + (TIME_TO_REAL(Sim_Timer.ET) / 1000.0) * Sim_Rate;
    ELSE
        Sim_Timer(IN := FALSE);
        Start_Sim_Weight := load_cell_value;
    END_IF;
END_IF;


(* 2. EMERGENCY STOP LOGIC (Error 12) *)
IF E_Stop_Active THEN
    FOR i := 1 TO 6 DO
        Auto_Bin[i] := FALSE;
        auto_bin_cutoff[i] := FALSE;
        auto_bin_motor[i] := FALSE;
    END_FOR;
    Sequence_Complete := FALSE;
    Active_Material_ID := 0;
    Active_Bin_ID := 0;
    Active_Target_Weight := 0.0;
    Error_Code := 12;
    Status_Message := 'Error 12: Emergency Stop Active!';
    Step := 99;
    Transition_Timer(IN := FALSE);
    Completion_Timer(IN := FALSE);
    RETURN;
END_IF;


(* 3. RECIPE SEQUENCE START *)
IF Step = 0 AND Start_Button THEN
    Step := 1;
    bin_last_weight := load_cell_value;
    Sequence_Complete := FALSE;
    Error_Code := 0;
    Status_Message := 'Auto Batch Started';
    Active_Target_Weight := 0.0;
    (* Clear actual weights and outputs on start *)
    FOR i := 1 TO 6 DO
        Actual_Weights[i] := 0.0;
        Auto_Bin[i] := FALSE;
        auto_bin_cutoff[i] := FALSE;
        auto_bin_motor[i] := FALSE;
    END_FOR;
END_IF;


(* 4. SEQUENCE CONTROL STATE MACHINE *)
CASE Step OF
    0:
        Active_Material_ID := 0;
        Active_Bin_ID := 0;
        Active_Target_Weight := 0.0;
        IF Error_Code = 0 THEN Status_Message := 'Auto Idle'; END_IF;
        
    1..6: (* Discharging Silos 1 to 6 *)
        Mat_Idx := Auto_Bin_Material_Mapping[Step];
        
        IF Mat_Idx = 0 THEN
            (* Skip this bin instantly *)
            Step := Step + 1;
        ELSE
            (* Fetch target weight from global Recipe_Weights array *)
            bin_set_value := GVL.Recipe_Weights[Mat_Idx];
            
            (* Calculate effective target weight (Looked up Target - Tolerance) *)
            target_act_bin := bin_set_value - Auto_Bin_Tolerance[Step];
            Active_Target_Weight := target_act_bin;
            
            (* Calculate weight added by current active bin *)
            actual_bin := load_cell_value - bin_last_weight;
            Actual_Weights[Step] := actual_bin;
            
            (* Calculate cutoff trigger threshold *)
            cutoff_trigger_weight := target_act_bin - Auto_Coarse_To_Fine_speed[Step];
            
            Active_Material_ID := Mat_Idx;
            Active_Bin_ID := Step;
            Status_Message := 'Auto Pouring';
            
            (* COARSE/FINE FEED TRANSITIONS WITH TOLERANCE OFFSETS *)
            IF actual_bin < cutoff_trigger_weight THEN
                (* Phase 1: Coarse Feed (Conveyor Motor ON, Main Valve ON, Fine Cutoff OFF) *)
                Auto_Bin[Step] := TRUE;
                auto_bin_cutoff[Step] := FALSE;
                auto_bin_motor[Step] := TRUE;
            ELSIF actual_bin < target_act_bin THEN
                (* Phase 2: Fine Feed (Conveyor Motor ON, Main Valve OFF, Fine Cutoff ON) *)
                Auto_Bin[Step] := FALSE;
                auto_bin_cutoff[Step] := TRUE;
                auto_bin_motor[Step] := TRUE;
            ELSE
                (* Phase 3: Completed (All OFF) *)
                Auto_Bin[Step] := FALSE;
                auto_bin_cutoff[Step] := FALSE;
                auto_bin_motor[Step] := FALSE;
                bin_last_weight := load_cell_value;
                Active_Target_Weight := 0.0;
                Step := 10 + Step; // Offset to separate transition states
            END_IF;
            
            (* RUNTIME CHECKS *)
            (* Check 21 & 22: Scale Limits *)
            IF load_cell_value > 500.0 THEN
                Error_Code := 21;
                Status_Message := 'Error 21: Scale Overloaded!';
                Step := 99;
                RETURN;
            ELSIF load_cell_value < 0.0 THEN
                Error_Code := 22;
                Status_Message := 'Error 22: Scale Underloaded/Fault!';
                Step := 99;
                RETURN;
            END_IF;
        END_IF;

    11..15: (* Transition Delays (Between Bins) *)
        Active_Material_ID := 0;
        Active_Bin_ID := 0;
        Active_Target_Weight := 0.0;
        Status_Message := 'Transition Delay';
        
        Transition_Timer(IN := TRUE, PT := Step_Delay_Time);
        IF Transition_Timer.Q THEN
            Transition_Timer(IN := FALSE);
            Step := (Step - 10) + 1; // Advance to next bin
        END_IF;
        
    16: (* Transition Delay After Last Bin (Bin 6) Closes *)
        Active_Material_ID := 0;
        Active_Bin_ID := 0;
        Active_Target_Weight := 0.0;
        Status_Message := 'Settling Last Bin';
        
        Transition_Timer(IN := TRUE, PT := Step_Delay_Time);
        IF Transition_Timer.Q THEN
            Transition_Timer(IN := FALSE);
            Step := 7; // Go to post-discharge wait step
        END_IF;

    7: (* Wait 2 Seconds After Closing the Last Bin *)
        Active_Material_ID := 0;
        Active_Bin_ID := 0;
        Active_Target_Weight := 0.0;
        Status_Message := 'Settling Delay';
        Completion_Timer(IN := TRUE, PT := Post_Complete_Delay);
        IF Completion_Timer.Q THEN
            Completion_Timer(IN := FALSE);
            Step := 8; // Proceed to reset last weight
        END_IF;
        
    8: (* Reset bin_last_weight to 0 & Complete *)
        Active_Material_ID := 0;
        Active_Bin_ID := 0;
        Active_Target_Weight := 0.0;
        Status_Message := 'Sequence Completed';
        bin_last_weight := 0.0;
        Sequence_Complete := TRUE;
        
        IF NOT Start_Button THEN
            Step := 0;
            Sequence_Complete := FALSE;
            (* Reset all actual weights at completion once start is released *)
            FOR i := 1 TO 6 DO
                Actual_Weights[i] := 0.0;
            END_FOR;
        END_IF;
        
    99: (* Error Abort state *)
        FOR i := 1 TO 6 DO 
            Auto_Bin[i] := FALSE; 
            auto_bin_cutoff[i] := FALSE;
            auto_bin_motor[i] := FALSE;
        END_FOR;
        Active_Material_ID := 0;
        Active_Bin_ID := 0;
        Active_Target_Weight := 0.0;
        IF NOT Start_Button THEN
            Step := 0;
            Error_Code := 0;
            Status_Message := 'Auto Idle';
        END_IF;
END_CASE;

END_FUNCTION_BLOCK

// PLC_AC500_V3/Application/old_version/Manual_Batching_V9
FUNCTION_BLOCK Manual_Batching_V9
VAR_INPUT
    Start_Button : BOOL;      // Signal to start the batching sequence
    E_Stop_Active : BOOL;     // Emergency Stop active signal
    Manual_Bin_Material_Mapping : ARRAY[1..10] OF INT; // Material index mapping for 10 manual silos
    Manual_Coarse_To_Fine_speed : ARRAY[1..10] OF REAL; // Cutoff weight thresholds (kg)
    Manual_Bin_Tolerance : ARRAY[1..10] OF REAL; // Tolerance weight offset values (kg)
END_VAR
VAR_IN_OUT
    load_cell_value : REAL;   // Weight value read/written from load cell
END_VAR
VAR_OUTPUT
    Manual_Bin : ARRAY[1..10] OF BOOL; // Prompts/indicators for Bins 7..16
    manual_bin_cutoff : ARRAY[1..10] OF BOOL; // Manual pre-cutoff indicators
    manual_bin_motor : ARRAY[1..10] OF BOOL; // Main manual feeder motor outputs
    Actual_Weights : ARRAY[1..10] OF REAL; // Actual weight poured per silo
    Sequence_Complete : BOOL;  // Batch complete flag
    Active_Material_ID : INT;  // Currently active ingredient ID
    Active_Bin_ID : INT;       // Currently active physical Bin ID (7..16)
    Active_Target_Weight : REAL; // Recipe target weight of active bin (with tolerance applied)
    Error_Code : INT;          // Active error code
    Status_Message : STRING;   // Diagnostic text message
END_VAR
VAR
    Step : INT := 0;          // State machine index (0: Idle, 1..10: Bins, 11..20: Delays, 30: Settling, 40: Complete, 99: Error)
    bin_last_weight : REAL;   // Baseline weight on the load cell before starting current bin
    actual_bin : REAL;        // Current weight added from active bin
    target_act_bin : REAL;    // Effective target weight to add from the active bin (GVL target - Tolerance)
    bin_set_value : REAL;     // Setpoint weight looked up from GVL
    cutoff_trigger_weight : REAL; // Calculated target threshold weight minus cutoff and tolerance values
    
    Mat_Idx : INT;
    i : INT;                  // General loop index
    
    (* TIMERS FOR TRANSITIONS & DELAYS *)
    Transition_Timer : TON;
    Completion_Timer : TON;
    Step_Delay_Time : TIME := T#2S;
    Post_Complete_Delay : TIME := T#2S;
    
    (* DIAGNOSTIC TIMERS *)
    Operator_Timer : TON;
    
    (* SELF-CONTAINED SIMULATION VARIABLES *)
    Simulation_Mode : BOOL := TRUE;
    Sim_Rate : REAL := 10.0;            // Simulated pouring speed (10.0 kg/s)
    Sim_Timer : TON;
    Start_Sim_Weight : REAL;
    Discharge_Active : BOOL;
END_VAR

(* Manual Batching FB V9 with Tolerance Logic *)

(* 1. SIMULATION WEIGHT MANAGEMENT *)
IF Simulation_Mode AND Step <> 99 THEN
    (* Reset simulation to baseline *)
    IF Step = 0 AND NOT Start_Button AND NOT Sequence_Complete THEN
        load_cell_value := 0.0;
        bin_last_weight := 0.0;
        Start_Sim_Weight := 0.0;
        Sim_Timer(IN := FALSE);
    END_IF;
    
    (* Check if operator is actively pouring *)
    Discharge_Active := FALSE;
    IF Step >= 1 AND Step <= 10 THEN
        Discharge_Active := manual_bin_motor[Step];
    END_IF;
    
    (* Simulate weight gain on the load cell *)
    IF Discharge_Active THEN
        Sim_Timer(IN := TRUE, PT := T#1000S);
        load_cell_value := Start_Sim_Weight + (TIME_TO_REAL(Sim_Timer.ET) / 1000.0) * Sim_Rate;
    ELSE
        Sim_Timer(IN := FALSE);
        Start_Sim_Weight := load_cell_value;
    END_IF;
END_IF;


(* 2. EMERGENCY STOP LOGIC (Error 12) *)
IF E_Stop_Active THEN
    FOR i := 1 TO 10 DO
        Manual_Bin[i] := FALSE;
        manual_bin_cutoff[i] := FALSE;
        manual_bin_motor[i] := FALSE;
    END_FOR;
    Sequence_Complete := FALSE;
    Active_Material_ID := 0;
    Active_Bin_ID := 0;
    Active_Target_Weight := 0.0;
    Error_Code := 12;
    Status_Message := 'Error 12: Emergency Stop Active!';
    Step := 99;
    Transition_Timer(IN := FALSE);
    Completion_Timer(IN := FALSE);
    RETURN;
END_IF;


(* 3. RECIPE SEQUENCE START *)
IF Step = 0 AND Start_Button THEN
    Step := 1;
    bin_last_weight := load_cell_value;
    Sequence_Complete := FALSE;
    Error_Code := 0;
    Status_Message := 'Manual Batch Started';
    Active_Target_Weight := 0.0;
    (* Clear actual weights on start *)
    FOR i := 1 TO 10 DO
        Actual_Weights[i] := 0.0;
        Manual_Bin[i] := FALSE;
        manual_bin_cutoff[i] := FALSE;
        manual_bin_motor[i] := FALSE;
    END_FOR;
END_IF;


(* 4. SEQUENCE CONTROL STATE MACHINE *)
CASE Step OF
    0:
        Active_Material_ID := 0;
        Active_Bin_ID := 0;
        Active_Target_Weight := 0.0;
        IF Error_Code = 0 THEN Status_Message := 'Manual Idle'; END_IF;
        
    1..10: (* Prompts Silos 7 to 16 *)
        Mat_Idx := Manual_Bin_Material_Mapping[Step];
        
        IF Mat_Idx = 0 THEN
            (* Skip this bin instantly *)
            Step := Step + 1;
        ELSE
            (* Fetch target weight from global Recipe_Weights array *)
            bin_set_value := GVL.Recipe_Weights[Mat_Idx];
            
            (* Calculate effective target weight (Looked up Target - Tolerance) *)
            target_act_bin := bin_set_value - Manual_Bin_Tolerance[Step];
            Active_Target_Weight := target_act_bin;
            
            (* Calculate weight added by current active bin *)
            actual_bin := load_cell_value - bin_last_weight;
            Actual_Weights[Step] := actual_bin;
            
            (* Calculate cutoff trigger threshold *)
            cutoff_trigger_weight := target_act_bin - Manual_Coarse_To_Fine_speed[Step];
            
            Active_Material_ID := Mat_Idx;
            Active_Bin_ID := Step;
            Status_Message := 'Manual Pouring Active';
            
            (* COARSE/FINE FEED TRANSITIONS WITH TOLERANCE OFFSETS *)
            IF actual_bin < cutoff_trigger_weight THEN
                (* Phase 1: Coarse Feed (Motor ON, Prompt ON, Cutoff OFF) *)
                Manual_Bin[Step] := TRUE;
                manual_bin_cutoff[Step] := FALSE;
                manual_bin_motor[Step] := TRUE;
            ELSIF actual_bin < target_act_bin THEN
                (* Phase 2: Fine Feed (Motor ON, Prompt OFF, Cutoff ON) *)
                Manual_Bin[Step] := FALSE;
                manual_bin_cutoff[Step] := TRUE;
                manual_bin_motor[Step] := TRUE;
            ELSE
                (* Phase 3: Completed (All OFF) *)
                Manual_Bin[Step] := FALSE;
                manual_bin_cutoff[Step] := FALSE;
                manual_bin_motor[Step] := FALSE;
                bin_last_weight := load_cell_value;
                Active_Target_Weight := 0.0;
                Step := 10 + Step; // Offset to separate transition states
            END_IF;
            
            (* RUNTIME CHECKS *)
            (* Check 21 & 22: Scale Limits *)
            IF load_cell_value > 500.0 THEN
                Error_Code := 21;
                Status_Message := 'Error 21: Scale Overloaded!';
                Step := 99;
                RETURN;
            ELSIF load_cell_value < 0.0 THEN
                Error_Code := 22;
                Status_Message := 'Error 22: Scale Underloaded/Fault!';
                Step := 99;
                RETURN;
            END_IF;
            
            (* Check 30: Operator Timeout *)
            Operator_Timer(IN := manual_bin_motor[Step], PT := T#300S);
            IF Operator_Timer.Q THEN
                Error_Code := 30;
                Status_Message := 'Error 30: Manual Operator Timeout!';
                Step := 99;
                RETURN;
            END_IF;
        END_IF;

    11..19: (* Transition Delays (Between Bins) *)
        Active_Material_ID := 0;
        Active_Bin_ID := 0;
        Active_Target_Weight := 0.0;
        Status_Message := 'Transition Delay';
        Transition_Timer(IN := TRUE, PT := Step_Delay_Time);
        IF Transition_Timer.Q THEN
            Transition_Timer(IN := FALSE);
            Step := (Step - 10) + 1; // Advance to next bin
        END_IF;
        
    20: (* Transition Delay After Last Bin (Bin 10) Closes *)
        Active_Material_ID := 0;
        Active_Bin_ID := 0;
        Active_Target_Weight := 0.0;
        Status_Message := 'Settling Last Bin';
        Transition_Timer(IN := TRUE, PT := Step_Delay_Time);
        IF Transition_Timer.Q THEN
            Transition_Timer(IN := FALSE);
            Step := 30; // Go to post-discharge wait step (State 30)
        END_IF;

    30: (* Wait 2 Seconds After Closing the Last Bin *)
        Active_Material_ID := 0;
        Active_Bin_ID := 0;
        Active_Target_Weight := 0.0;
        Status_Message := 'Settling Delay';
        Completion_Timer(IN := TRUE, PT := Post_Complete_Delay);
        IF Completion_Timer.Q THEN
            Completion_Timer(IN := FALSE);
            Step := 40; // Proceed to reset last weight (State 40)
        END_IF;
        
    40: (* Reset bin_last_weight to 0 & Complete *)
        Active_Material_ID := 0;
        Active_Bin_ID := 0;
        Active_Target_Weight := 0.0;
        Status_Message := 'Sequence Completed';
        bin_last_weight := 0.0;
        Sequence_Complete := TRUE;
        
        IF NOT Start_Button THEN
            Step := 0;
            Sequence_Complete := FALSE;
            (* Reset all actual weights at completion once start is released *)
            FOR i := 1 TO 10 DO
                Actual_Weights[i] := 0.0;
            END_FOR;
        END_IF;
        
    99: (* Error Abort state *)
        FOR i := 1 TO 10 DO 
            Manual_Bin[i] := FALSE;
            manual_bin_cutoff[i] := FALSE;
            manual_bin_motor[i] := FALSE;
        END_FOR;
        Active_Material_ID := 0;
        Active_Bin_ID := 0;
        Active_Target_Weight := 0.0;
        IF NOT Start_Button THEN
            Step := 0;
            Error_Code := 0;
            Status_Message := 'Manual Idle';
        END_IF;
END_CASE;

END_FUNCTION_BLOCK

// PLC_AC500_V3/Application/old_version/batching9
PROGRAM batching9
VAR
    Auto_Ctrl : Auto_Batching_V9;
    Manual_Ctrl : Manual_Batching_V9;
    
    (* Global Inputs & Toggles *)
    Start_Button : BOOL;
    E_Stop_Active : BOOL;
    
    (* Parallel Weight Feedbacks *)
    load_cell_auto : REAL;
    load_cell_manual : REAL;
    
    (* Sub-Block Diagnostic Indicators - Ordered exactly below loadcell *)
    Auto_Active_Mat : INT;
    Auto_Active_Bin : INT;
    Auto_Active_Target : REAL; // Active Target Weight for Auto (displays GVL setpoint - Tolerance)
    Auto_Err : INT;
    Auto_Msg : STRING;
    
    Manual_Active_Mat : INT;
    Manual_Active_Bin : INT;
    Manual_Active_Target : REAL; // Active Target Weight for Manual (displays GVL setpoint - Tolerance)
    Manual_Err : INT;
    Manual_Msg : STRING;
    
    (* Process Outputs *)
    Auto_Bin : ARRAY[1..6] OF BOOL; // Valve control outputs (Coarse)
    auto_bin_cutoff : ARRAY[1..6] OF BOOL; // Cutoff indicators (Fine)
    auto_bin_motor : ARRAY[1..6] OF BOOL; // Conveyor/feeder motor outputs
    
    Manual_Bin : ARRAY[1..10] OF BOOL; // Prompt indicators (Coarse)
    manual_bin_cutoff : ARRAY[1..10] OF BOOL; // Cutoff indicators (Fine)
    manual_bin_motor : ARRAY[1..10] OF BOOL; // Conveyor/feeder motor outputs
    
    Auto_Weights : ARRAY[1..6] OF REAL;
    Manual_Weights : ARRAY[1..10] OF REAL;
    
    Auto_Complete : BOOL;
    Manual_Complete : BOOL;
    Sequence_Complete : BOOL;
    
    (* Diagnostics & Interlocks *)
    Error_Code : INT := 0;
    Status_Message : STRING := 'System Ready';
    
    (* Array Configurations & Mapping - Renamed for clarity *)
    Auto_Bin_Material_Mapping : ARRAY[1..6] OF INT := [1, 2, 0, 4, 5, 6];
    Manual_Bin_Material_Mapping : ARRAY[1..10] OF INT := [7, 8, 0, 10, 11, 12, 13, 14, 15, 16];
    Auto_Coarse_To_Fine_speed : ARRAY[1..6] OF REAL := [2.0, 1.5, 0.0, 3.0, 5.0, 1.0]; // Cutoff margins (kg)
    Manual_Coarse_To_Fine_speed : ARRAY[1..10] OF REAL := [2.0, 1.5, 0.0, 3.0, 5.0, 1.0, 2.0, 2.0, 2.0, 2.0];
    Auto_Bin_Tolerance : ARRAY[1..6] OF REAL := [1.0, 0.5, 0.0, 1.0, 2.0, 0.5]; // Tolerance offsets (kg)
    Manual_Bin_Tolerance : ARRAY[1..10] OF REAL := [1.0, 0.5, 0.0, 1.0, 2.0, 0.5, 1.0, 1.0, 1.0, 1.0];
    
    i : INT;
    j : INT;
    Duplicate_Found : BOOL;
    Invalid_Material_Range : BOOL;
    Zero_Target_Found : BOOL;
    Conf_Err_Id : INT;
END_VAR

(* 1. STARTUP CONFIGURATION CHECKS *)
Duplicate_Found := FALSE;
Invalid_Material_Range := FALSE;
Zero_Target_Found := FALSE;

FOR i := 1 TO 6 DO
    (* Check 2: Out of Range (Auto) *)
    IF Auto_Bin_Material_Mapping[i] < 0 OR Auto_Bin_Material_Mapping[i] > 20 THEN
        Invalid_Material_Range := TRUE;
    END_IF;
    
    (* Check 3: Zero Target (Auto) *)
    IF Auto_Bin_Material_Mapping[i] <> 0 AND Auto_Bin_Material_Mapping[i] <= 20 THEN
        IF GVL.Recipe_Weights[Auto_Bin_Material_Mapping[i]] = 0.0 THEN
            Zero_Target_Found := TRUE;
        END_IF;
    END_IF;
    
    (* Check 1: Duplicate Cross-Array Material ID *)
    IF Auto_Bin_Material_Mapping[i] <> 0 AND Auto_Bin_Material_Mapping[i] <= 20 THEN
        FOR j := 1 TO 10 DO
            IF Auto_Bin_Material_Mapping[i] = Manual_Bin_Material_Mapping[j] THEN
                Duplicate_Found := TRUE;
            END_IF;
        END_FOR;
    END_IF;
END_FOR;

FOR j := 1 TO 10 DO
    (* Check 2: Out of Range (Manual) *)
    IF Manual_Bin_Material_Mapping[j] < 0 OR Manual_Bin_Material_Mapping[j] > 20 THEN
        Invalid_Material_Range := TRUE;
    END_IF;
    
    (* Check 3: Zero Target (Manual) *)
    IF Manual_Bin_Material_Mapping[j] <> 0 AND Manual_Bin_Material_Mapping[j] <= 20 THEN
        IF GVL.Recipe_Weights[Manual_Bin_Material_Mapping[j]] = 0.0 THEN
            Zero_Target_Found := TRUE;
        END_IF;
    END_IF;
END_FOR;

(* Configuration Error Resolution *)
IF Duplicate_Found THEN
    Error_Code := 1;
    Status_Message := 'Error 1: Duplicate Material ID mapped in Auto and Manual!';
ELSIF Invalid_Material_Range THEN
    Error_Code := 2;
    Status_Message := 'Error 2: Material Index configuration out of range (1..20)!';
ELSIF Zero_Target_Found THEN
    Error_Code := 3;
    Status_Message := 'Error 3: Configured Material ID has a 0.0 kg target weight!';
ELSE
    IF Error_Code <= 3 THEN
        Error_Code := 0;
    END_IF;
END_IF;

(* Abort sequences if a configuration error exists *)
IF Error_Code >= 1 AND Error_Code <= 3 THEN
    FOR i := 1 TO 6 DO Auto_Bin[i] := FALSE; auto_bin_cutoff[i] := FALSE; auto_bin_motor[i] := FALSE; END_FOR;
    FOR i := 1 TO 10 DO Manual_Bin[i] := FALSE; manual_bin_cutoff[i] := FALSE; manual_bin_motor[i] := FALSE; END_FOR;
    Auto_Ctrl(Start_Button := FALSE, E_Stop_Active := TRUE, load_cell_value := load_cell_auto);
    Manual_Ctrl(Start_Button := FALSE, E_Stop_Active := TRUE, load_cell_value := load_cell_manual);
    Auto_Active_Target := 0.0;
    Manual_Active_Target := 0.0;
    RETURN;
END_IF;


(* 2. CONCURRENT EXECUTION OF FB INSTANCES *)
Auto_Ctrl(
    Start_Button := Start_Button,
    E_Stop_Active := E_Stop_Active,
    load_cell_value := load_cell_auto,
    Auto_Bin_Material_Mapping := Auto_Bin_Material_Mapping,
    Auto_Coarse_To_Fine_speed := Auto_Coarse_To_Fine_speed,
    Auto_Bin_Tolerance := Auto_Bin_Tolerance,
    Auto_Bin => Auto_Bin,
    auto_bin_cutoff => auto_bin_cutoff,
    auto_bin_motor => auto_bin_motor,
    Actual_Weights => Auto_Weights,
    Sequence_Complete => Auto_Complete,
    Active_Material_ID => Auto_Active_Mat,
    Active_Bin_ID => Auto_Active_Bin,
    Active_Target_Weight => Auto_Active_Target,
    Error_Code => Auto_Err,
    Status_Message => Auto_Msg
);

Manual_Ctrl(
    Start_Button := Start_Button,
    E_Stop_Active := E_Stop_Active,
    load_cell_value := load_cell_manual,
    Manual_Bin_Material_Mapping := Manual_Bin_Material_Mapping,
    Manual_Coarse_To_Fine_speed := Manual_Coarse_To_Fine_speed,
    Manual_Bin_Tolerance := Manual_Bin_Tolerance,
    Manual_Bin => Manual_Bin,
    manual_bin_cutoff => manual_bin_cutoff,
    manual_bin_motor => manual_bin_motor,
    Actual_Weights => Manual_Weights,
    Sequence_Complete => Manual_Complete,
    Active_Material_ID => Manual_Active_Mat,
    Active_Bin_ID => Manual_Active_Bin,
    Active_Target_Weight => Manual_Active_Target,
    Error_Code => Manual_Err,
    Status_Message => Manual_Msg
);

(* Runtime Error Mapping & Aggregation *)
IF Auto_Err <> 0 THEN
    Error_Code := Auto_Err;
    Status_Message := CONCAT('Auto Error: ', Auto_Msg);
ELSIF Manual_Err <> 0 THEN
    Error_Code := Manual_Err;
    Status_Message := CONCAT('Manual Error: ', Manual_Msg);
ELSE
    Error_Code := 0;
    
    Sequence_Complete := Auto_Complete AND Manual_Complete;
    IF Sequence_Complete THEN
        Status_Message := 'Batch Sequence Completed';
    ELSIF Start_Button THEN
        Status_Message := 'Batch Sequence Running';
    ELSE
        Status_Message := 'System Ready';
    END_IF;
END_IF;

END_PROGRAM

// PLC_AC500_V3/Application/old_version/Auto_Batching_V10
FUNCTION_BLOCK Auto_Batching_V10
VAR_INPUT
    Start_Button : BOOL;      // Signal to start the batching sequence
    E_Stop_Active : BOOL;     // Emergency Stop active signal
    Auto_Bin_Material_Mapping : ARRAY[1..6] OF INT; // Material index mapping for 6 bins
    Auto_Coarse_To_Fine_speed : ARRAY[1..6] OF REAL; // Cutoff weight thresholds (kg)
    Auto_Bin_Tolerance : ARRAY[1..6] OF REAL; // Tolerance weight offset values (kg)
END_VAR
VAR_IN_OUT
    load_cell_value : REAL;   // Weight value read/written from load cell
END_VAR
VAR_OUTPUT
    Auto_Bin : ARRAY[1..6] OF BOOL; // Coarse feed valve outputs
    auto_bin_cutoff : ARRAY[1..6] OF BOOL; // Fine feed cutoff trigger indicators
    auto_bin_motor : ARRAY[1..6] OF BOOL; // Main conveyor motor outputs
    Actual_Weights : ARRAY[1..6] OF REAL; // Actual weight poured per silo
    Sequence_Complete : BOOL;  // Batch complete flag
    Active_Material_ID : INT;  // Currently active ingredient ID
    Active_Bin_ID : INT;       // Currently active physical Bin ID (1..6)
    Active_Target_Weight : REAL; // Recipe target weight of active bin (with tolerance applied)
    Error_Code : INT;          // Active error code
    Status_Message : STRING;   // Diagnostic text message
END_VAR
VAR
    Step : INT := 0;          // State machine index (0: Idle, 1..6: Bins, 11..16: Delays, 7: Settling, 8: Complete, 99: Error)
    bin_last_weight : REAL;   // Baseline weight on the load cell before starting current bin
    actual_bin : REAL;        // Current weight added from active bin
    target_act_bin : REAL;    // Effective target weight to add from the active bin (GVL target - Tolerance)
    cutoff_trigger_weight : REAL; // Calculated trigger weight (target - Tolerance - Cutoff)
    
    Mat_Idx : INT;
    i : INT;                  // General loop index
    
    (* TIMERS FOR TRANSITIONS & DELAYS *)
    Transition_Timer : TON;
    Completion_Timer : TON;
    Step_Delay_Time : TIME := T#2S;
    Post_Complete_Delay : TIME := T#2S;
    
    (* SELF-CONTAINED SIMULATION VARIABLES *)
    Simulation_Mode : BOOL := TRUE;
    Sim_Rate : REAL := 10.0;            // Simulated pouring speed (10.0 kg/s)
    Sim_Timer : TON;
    Start_Sim_Weight : REAL;
    Discharge_Active : BOOL;
END_VAR

(* Auto Batching FB V10 with Tolerance Logic & Skipping / E-Stop Fixes *)

(* 1. SELF-CONTAINED SIMULATION WEIGHT MANAGEMENT *)
IF Simulation_Mode AND Step <> 99 THEN
    (* Reset simulation to baseline *)
    IF Step = 0 AND NOT Start_Button AND NOT Sequence_Complete THEN
        load_cell_value := 0.0;
        bin_last_weight := 0.0;
        Start_Sim_Weight := 0.0;
        Sim_Timer(IN := FALSE);
    END_IF;
    
    (* Check if any valve is actively discharging *)
    Discharge_Active := FALSE;
    IF Step >= 1 AND Step <= 6 THEN
        Discharge_Active := auto_bin_motor[Step];
    END_IF;
    
    (* Simulate weight gain on the load cell *)
    IF Discharge_Active THEN
        Sim_Timer(IN := TRUE, PT := T#1000S);
        load_cell_value := Start_Sim_Weight + (TIME_TO_REAL(Sim_Timer.ET) / 1000.0) * Sim_Rate;
    ELSE
        Sim_Timer(IN := FALSE);
        Start_Sim_Weight := load_cell_value;
    END_IF;
END_IF;


(* 2. EMERGENCY STOP LOGIC (Error 12) *)
IF E_Stop_Active THEN
    FOR i := 1 TO 6 DO
        Auto_Bin[i] := FALSE;
        auto_bin_cutoff[i] := FALSE;
        auto_bin_motor[i] := FALSE;
    END_FOR;
    Sequence_Complete := FALSE;
    Active_Material_ID := 0;
    Active_Bin_ID := 0;
    Active_Target_Weight := 0.0;
    Error_Code := 12;
    Status_Message := 'Error 12: Emergency Stop Active!';
    Step := 99;
    Transition_Timer(IN := FALSE);
    Completion_Timer(IN := FALSE);
    RETURN;
END_IF;


(* 3. RECIPE SEQUENCE START *)
IF Step = 0 AND Start_Button THEN
    Step := 1;
    bin_last_weight := load_cell_value;
    Sequence_Complete := FALSE;
    Error_Code := 0;
    Status_Message := 'Auto Batch Started';
    Active_Target_Weight := 0.0;
    (* Clear actual weights and outputs on start *)
    FOR i := 1 TO 6 DO
        Actual_Weights[i] := 0.0;
        Auto_Bin[i] := FALSE;
        auto_bin_cutoff[i] := FALSE;
        auto_bin_motor[i] := FALSE;
    END_FOR;
END_IF;


(* 4. SEQUENCE CONTROL STATE MACHINE *)
CASE Step OF
    0:
        Active_Material_ID := 0;
        Active_Bin_ID := 0;
        Active_Target_Weight := 0.0;
        IF Error_Code = 0 THEN Status_Message := 'Auto Idle'; END_IF;
        
    1..6: (* Discharging Silos 1 to 6 *)
        Mat_Idx := Auto_Bin_Material_Mapping[Step];
        
        (* Skip this step instantly if material mapping is 0 OR target weight is 0.0 kg *)
        IF Mat_Idx = 0 OR (Mat_Idx <= 20 AND GVL.Recipe_Weights[Mat_Idx] = 0.0) THEN
            Step := Step + 1;
        ELSE
            (* Calculate effective target weight (Looked up Target - Tolerance) *)
            target_act_bin := GVL.Recipe_Weights[Mat_Idx] - Auto_Bin_Tolerance[Step];
            Active_Target_Weight := target_act_bin;
            
            (* Calculate weight added by current active bin *)
            actual_bin := load_cell_value - bin_last_weight;
            Actual_Weights[Step] := actual_bin;
            
            (* Calculate cutoff trigger threshold *)
            cutoff_trigger_weight := target_act_bin - Auto_Coarse_To_Fine_speed[Step];
            
            Active_Material_ID := Mat_Idx;
            Active_Bin_ID := Step;
            Status_Message := 'Auto Pouring';
            
            (* COARSE/FINE FEED TRANSITIONS WITH TOLERANCE OFFSETS *)
            IF actual_bin < cutoff_trigger_weight THEN
                (* Phase 1: Coarse Feed (Conveyor Motor ON, Main Valve ON, Fine Cutoff OFF) *)
                Auto_Bin[Step] := TRUE;
                auto_bin_cutoff[Step] := FALSE;
                auto_bin_motor[Step] := TRUE;
            ELSIF actual_bin < target_act_bin THEN
                (* Phase 2: Fine Feed (Conveyor Motor ON, Main Valve OFF, Fine Cutoff ON) *)
                Auto_Bin[Step] := FALSE;
                auto_bin_cutoff[Step] := TRUE;
                auto_bin_motor[Step] := TRUE;
            ELSE
                (* Phase 3: Completed (All OFF) *)
                Auto_Bin[Step] := FALSE;
                auto_bin_cutoff[Step] := FALSE;
                auto_bin_motor[Step] := FALSE;
                bin_last_weight := load_cell_value;
                Active_Target_Weight := 0.0;
                Step := 10 + Step; // Offset to separate transition states
            END_IF;
            
            (* RUNTIME CHECKS *)
            (* Check 21 & 22: Scale Limits *)
            IF load_cell_value > 500.0 THEN
                Error_Code := 21;
                Status_Message := 'Error 21: Scale Overloaded!';
                Step := 99;
                RETURN;
            ELSIF load_cell_value < 0.0 THEN
                Error_Code := 22;
                Status_Message := 'Error 22: Scale Underloaded/Fault!';
                Step := 99;
                RETURN;
            END_IF;
        END_IF;

    11..15: (* Transition Delays (Between Bins) *)
        Active_Material_ID := 0;
        Active_Bin_ID := 0;
        Active_Target_Weight := 0.0;
        Status_Message := 'Transition Delay';
        
        Transition_Timer(IN := TRUE, PT := Step_Delay_Time);
        IF Transition_Timer.Q THEN
            Transition_Timer(IN := FALSE);
            Step := (Step - 10) + 1; // Advance to next bin
        END_IF;
        
    16: (* Transition Delay After Last Bin (Bin 6) Closes *)
        Active_Material_ID := 0;
        Active_Bin_ID := 0;
        Active_Target_Weight := 0.0;
        Status_Message := 'Settling Last Bin';
        
        Transition_Timer(IN := TRUE, PT := Step_Delay_Time);
        IF Transition_Timer.Q THEN
            Transition_Timer(IN := FALSE);
            Step := 7; // Go to post-discharge wait step
        END_IF;

    7: (* Wait 2 Seconds After Closing the Last Bin *)
        Active_Material_ID := 0;
        Active_Bin_ID := 0;
        Active_Target_Weight := 0.0;
        Status_Message := 'Settling Delay';
        Completion_Timer(IN := TRUE, PT := Post_Complete_Delay);
        IF Completion_Timer.Q THEN
            Completion_Timer(IN := FALSE);
            Step := 8; // Proceed to reset last weight
        END_IF;
        
    8: (* Reset bin_last_weight to 0 & Complete *)
        Active_Material_ID := 0;
        Active_Bin_ID := 0;
        Active_Target_Weight := 0.0;
        Status_Message := 'Sequence Completed';
        bin_last_weight := 0.0;
        Sequence_Complete := TRUE;
        
        IF NOT Start_Button THEN
            Step := 0;
            Sequence_Complete := FALSE;
            (* Reset all actual weights at completion once start is released *)
            FOR i := 1 TO 6 DO
                Actual_Weights[i] := 0.0;
            END_FOR;
        END_IF;
        
    99: (* Error Abort state *)
        FOR i := 1 TO 6 DO 
            Auto_Bin[i] := FALSE; 
            auto_bin_cutoff[i] := FALSE;
            auto_bin_motor[i] := FALSE;
        END_FOR;
        Active_Material_ID := 0;
        Active_Bin_ID := 0;
        Active_Target_Weight := 0.0;
        
        (* Prevent reset loop by checking E_Stop_Active *)
        IF NOT Start_Button AND NOT E_Stop_Active THEN
            Step := 0;
            Error_Code := 0;
            Status_Message := 'Auto Idle';
        END_IF;
END_CASE;

END_FUNCTION_BLOCK

// PLC_AC500_V3/Application/old_version/Manual_Batching_V10
FUNCTION_BLOCK Manual_Batching_V10
VAR_INPUT
    Start_Button : BOOL;      // Signal to start the batching sequence
    E_Stop_Active : BOOL;     // Emergency Stop active signal
    Manual_Bin_Material_Mapping : ARRAY[1..10] OF INT; // Material index mapping for 10 manual silos
    Manual_Coarse_To_Fine_speed : ARRAY[1..10] OF REAL; // Cutoff weight thresholds (kg)
    Manual_Bin_Tolerance : ARRAY[1..10] OF REAL; // Tolerance weight offset values (kg)
END_VAR
VAR_IN_OUT
    load_cell_value : REAL;   // Weight value read/written from load cell
END_VAR
VAR_OUTPUT
    Manual_Bin : ARRAY[1..10] OF BOOL; // Prompts/indicators for Bins 7..16
    manual_bin_cutoff : ARRAY[1..10] OF BOOL; // Manual pre-cutoff indicators
    manual_bin_motor : ARRAY[1..10] OF BOOL; // Main manual feeder motor outputs
    Actual_Weights : ARRAY[1..10] OF REAL; // Actual weight poured per silo
    Sequence_Complete : BOOL;  // Batch complete flag
    Active_Material_ID : INT;  // Currently active ingredient ID
    Active_Bin_ID : INT;       // Currently active physical Bin ID (7..16)
    Active_Target_Weight : REAL; // Recipe target weight of active bin (with tolerance applied)
    Error_Code : INT;          // Active error code
    Status_Message : STRING;   // Diagnostic text message
END_VAR
VAR
    Step : INT := 0;          // State machine index (0: Idle, 1..10: Bins, 11..20: Delays, 30: Settling, 40: Complete, 99: Error)
    bin_last_weight : REAL;   // Baseline weight on the load cell before starting current bin
    actual_bin : REAL;        // Current weight added from active bin
    target_act_bin : REAL;    // Effective target weight to add from the active bin (GVL target - Tolerance)
    cutoff_trigger_weight : REAL; // Calculated target threshold weight minus cutoff and tolerance values
    
    Mat_Idx : INT;
    i : INT;                  // General loop index
    
    (* TIMERS FOR TRANSITIONS & DELAYS *)
    Transition_Timer : TON;
    Completion_Timer : TON;
    Step_Delay_Time : TIME := T#2S;
    Post_Complete_Delay : TIME := T#2S;
    
    (* DIAGNOSTIC TIMERS *)
    Operator_Timer : TON;
    
    (* SELF-CONTAINED SIMULATION VARIABLES *)
    Simulation_Mode : BOOL := TRUE;
    Sim_Rate : REAL := 10.0;            // Simulated pouring speed (10.0 kg/s)
    Sim_Timer : TON;
    Start_Sim_Weight : REAL;
    Discharge_Active : BOOL;
END_VAR

(* Manual Batching FB V10 with Tolerance Logic & Skipping / E-Stop Fixes *)

(* 1. SIMULATION WEIGHT MANAGEMENT *)
IF Simulation_Mode AND Step <> 99 THEN
    (* Reset simulation to baseline *)
    IF Step = 0 AND NOT Start_Button AND NOT Sequence_Complete THEN
        load_cell_value := 0.0;
        bin_last_weight := 0.0;
        Start_Sim_Weight := 0.0;
        Sim_Timer(IN := FALSE);
    END_IF;
    
    (* Check if operator is actively pouring *)
    Discharge_Active := FALSE;
    IF Step >= 1 AND Step <= 10 THEN
        Discharge_Active := manual_bin_motor[Step];
    END_IF;
    
    (* Simulate weight gain on the load cell *)
    IF Discharge_Active THEN
        Sim_Timer(IN := TRUE, PT := T#1000S);
        load_cell_value := Start_Sim_Weight + (TIME_TO_REAL(Sim_Timer.ET) / 1000.0) * Sim_Rate;
    ELSE
        Sim_Timer(IN := FALSE);
        Start_Sim_Weight := load_cell_value;
    END_IF;
END_IF;


(* 2. EMERGENCY STOP LOGIC (Error 12) *)
IF E_Stop_Active THEN
    FOR i := 1 TO 10 DO
        Manual_Bin[i] := FALSE;
        manual_bin_cutoff[i] := FALSE;
        manual_bin_motor[i] := FALSE;
    END_FOR;
    Sequence_Complete := FALSE;
    Active_Material_ID := 0;
    Active_Bin_ID := 0;
    Active_Target_Weight := 0.0;
    Error_Code := 12;
    Status_Message := 'Error 12: Emergency Stop Active!';
    Step := 99;
    Transition_Timer(IN := FALSE);
    Completion_Timer(IN := FALSE);
    RETURN;
END_IF;


(* 3. RECIPE SEQUENCE START *)
IF Step = 0 AND Start_Button THEN
    Step := 1;
    bin_last_weight := load_cell_value;
    Sequence_Complete := FALSE;
    Error_Code := 0;
    Status_Message := 'Manual Batch Started';
    Active_Target_Weight := 0.0;
    (* Clear actual weights on start *)
    FOR i := 1 TO 10 DO
        Actual_Weights[i] := 0.0;
        Manual_Bin[i] := FALSE;
        manual_bin_cutoff[i] := FALSE;
        manual_bin_motor[i] := FALSE;
    END_FOR;
END_IF;


(* 4. SEQUENCE CONTROL STATE MACHINE *)
CASE Step OF
    0:
        Active_Material_ID := 0;
        Active_Bin_ID := 0;
        Active_Target_Weight := 0.0;
        IF Error_Code = 0 THEN Status_Message := 'Manual Idle'; END_IF;
        
    1..10: (* Prompts Silos 7 to 16 *)
        Mat_Idx := Manual_Bin_Material_Mapping[Step];
        
        (* Skip this step instantly if material mapping is 0 OR target weight is 0.0 kg *)
        IF Mat_Idx = 0 OR (Mat_Idx <= 20 AND GVL.Recipe_Weights[Mat_Idx] = 0.0) THEN
            Step := Step + 1;
        ELSE
            (* Calculate effective target weight (Looked up Target - Tolerance) *)
            target_act_bin := GVL.Recipe_Weights[Mat_Idx] - Manual_Bin_Tolerance[Step];
            Active_Target_Weight := target_act_bin;
            
            (* Calculate weight added by current active bin *)
            actual_bin := load_cell_value - bin_last_weight;
            Actual_Weights[Step] := actual_bin;
            
            (* Calculate cutoff trigger threshold *)
            cutoff_trigger_weight := target_act_bin - Manual_Coarse_To_Fine_speed[Step];
            
            Active_Material_ID := Mat_Idx;
            Active_Bin_ID := Step;
            Status_Message := 'Manual Pouring Active';
            
            (* COARSE/FINE FEED TRANSITIONS WITH TOLERANCE OFFSETS *)
            IF actual_bin < cutoff_trigger_weight THEN
                (* Phase 1: Coarse Feed (Motor ON, Prompt ON, Cutoff OFF) *)
                Manual_Bin[Step] := TRUE;
                manual_bin_cutoff[Step] := FALSE;
                manual_bin_motor[Step] := TRUE;
            ELSIF actual_bin < target_act_bin THEN
                (* Phase 2: Fine Feed (Motor ON, Prompt OFF, Cutoff ON) *)
                Manual_Bin[Step] := FALSE;
                manual_bin_cutoff[Step] := TRUE;
                manual_bin_motor[Step] := TRUE;
            ELSE
                (* Phase 3: Completed (All OFF) *)
                Manual_Bin[Step] := FALSE;
                manual_bin_cutoff[Step] := FALSE;
                manual_bin_motor[Step] := FALSE;
                bin_last_weight := load_cell_value;
                Active_Target_Weight := 0.0;
                Step := 10 + Step; // Offset to separate transition states
            END_IF;
            
            (* RUNTIME CHECKS *)
            (* Check 21 & 22: Scale Limits *)
            IF load_cell_value > 500.0 THEN
                Error_Code := 21;
                Status_Message := 'Error 21: Scale Overloaded!';
                Step := 99;
                RETURN;
            ELSIF load_cell_value < 0.0 THEN
                Error_Code := 22;
                Status_Message := 'Error 22: Scale Underloaded/Fault!';
                Step := 99;
                RETURN;
            END_IF;
            
            (* Check 30: Operator Timeout *)
            Operator_Timer(IN := manual_bin_motor[Step], PT := T#300S);
            IF Operator_Timer.Q THEN
                Error_Code := 30;
                Status_Message := 'Error 30: Manual Operator Timeout!';
                Step := 99;
                RETURN;
            END_IF;
        END_IF;

    11..19: (* Transition Delays (Between Bins) *)
        Active_Material_ID := 0;
        Active_Bin_ID := 0;
        Active_Target_Weight := 0.0;
        Status_Message := 'Transition Delay';
        Transition_Timer(IN := TRUE, PT := Step_Delay_Time);
        IF Transition_Timer.Q THEN
            Transition_Timer(IN := FALSE);
            Step := (Step - 10) + 1; // Advance to next bin
        END_IF;
        
